				MB_BitStato[192]:=ModBus.MB_MASTER.ReceiveBuffer.Data[3].0; (*Vedi Tabella *)
				MB_BitStato[193]:=ModBus.MB_MASTER.ReceiveBuffer.Data[3].1; (*Vedi Tabella *)
				MB_BitStato[194]:=ModBus.MB_MASTER.ReceiveBuffer.Data[3].2; (*Vedi Tabella *)
				MB_BitStato[195]:=ModBus.MB_MASTER.ReceiveBuffer.Data[3].3; (*Vedi Tabella *)
				MB_BitStato[196]:=ModBus.MB_MASTER.ReceiveBuffer.Data[3].4; (*Vedi Tabella *)
				MB_BitStato[197]:=ModBus.MB_MASTER.ReceiveBuffer.Data[3].5; (*Vedi Tabella *)
				MB_BitStato[198]:=ModBus.MB_MASTER.ReceiveBuffer.Data[3].6; (*Vedi Tabella *)
				MB_BitStato[199]:=ModBus.MB_MASTER.ReceiveBuffer.Data[3].7; (*Vedi Tabella *)
				MB_BitStato[200]:=ModBus.MB_MASTER.ReceiveBuffer.Data[4].0; (*Vedi Tabella *)
				MB_BitStato[201]:=ModBus.MB_MASTER.ReceiveBuffer.Data[4].1; (*Vedi Tabella *)
				MB_BitStato[202]:=ModBus.MB_MASTER.ReceiveBuffer.Data[4].2; (*Vedi Tabella *)
				MB_BitStato[203]:=ModBus.MB_MASTER.ReceiveBuffer.Data[4].3; (*Vedi Tabella *)
				MB_BitStato[204]:=ModBus.MB_MASTER.ReceiveBuffer.Data[4].4; (*Vedi Tabella *)
				MB_BitStato[205]:=ModBus.MB_MASTER.ReceiveBuffer.Data[4].5; (*Vedi Tabella *)
				MB_BitStato[206]:=ModBus.MB_MASTER.ReceiveBuffer.Data[4].6; (*Vedi Tabella *)
				MB_BitStato[207]:=ModBus.MB_MASTER.ReceiveBuffer.Data[4].7; (*Vedi Tabella *)
				MB_BitStato[208]:=ModBus.MB_MASTER.ReceiveBuffer.Data[5].0; (*Vedi Tabella *)
				MB_BitStato[209]:=ModBus.MB_MASTER.ReceiveBuffer.Data[5].1; (*Vedi Tabella *)
				MB_BitStato[210]:=ModBus.MB_MASTER.ReceiveBuffer.Data[5].2; (*Vedi Tabella *)
				MB_BitStato[211]:=ModBus.MB_MASTER.ReceiveBuffer.Data[5].3; (*Vedi Tabella *)
				MB_BitStato[212]:=ModBus.MB_MASTER.ReceiveBuffer.Data[5].4; (*Vedi Tabella *)
				MB_BitStato[213]:=ModBus.MB_MASTER.ReceiveBuffer.Data[5].5; (*Vedi Tabella *)
				MB_BitStato[214]:=ModBus.MB_MASTER.ReceiveBuffer.Data[5].6; (*Vedi Tabella *)
				MB_BitStato[215]:=ModBus.MB_MASTER.ReceiveBuffer.Data[5].7; (*Vedi Tabella *)
				MB_BitStato[216]:=ModBus.MB_MASTER.ReceiveBuffer.Data[6].0; (*Vedi Tabella *)
				MB_BitStato[217]:=ModBus.MB_MASTER.ReceiveBuffer.Data[6].1; (*Vedi Tabella *)
				MB_BitStato[218]:=ModBus.MB_MASTER.ReceiveBuffer.Data[6].2; (*Vedi Tabella *)
				MB_BitStato[219]:=ModBus.MB_MASTER.ReceiveBuffer.Data[6].3; (*Vedi Tabella *)
				MB_BitStato[220]:=ModBus.MB_MASTER.ReceiveBuffer.Data[6].4; (*Vedi Tabella *)
				MB_BitStato[221]:=ModBus.MB_MASTER.ReceiveBuffer.Data[6].5; (*Vedi Tabella *)
				MB_BitStato[222]:=ModBus.MB_MASTER.ReceiveBuffer.Data[6].6; (*Vedi Tabella *)
				MB_BitStato[223]:=ModBus.MB_MASTER.ReceiveBuffer.Data[6].7; (*Vedi Tabella *)
				MB_BitStato[224]:=ModBus.MB_MASTER.ReceiveBuffer.Data[7].0; (*Vedi Tabella *)
				MB_BitStato[225]:=ModBus.MB_MASTER.ReceiveBuffer.Data[7].1; (*Vedi Tabella *)
				MB_BitStato[226]:=ModBus.MB_MASTER.ReceiveBuffer.Data[7].2; (*Vedi Tabella *)
				MB_BitStato[227]:=ModBus.MB_MASTER.ReceiveBuffer.Data[7].3; (*Vedi Tabella *)
				MB_BitStato[228]:=ModBus.MB_MASTER.ReceiveBuffer.Data[7].4; (*Vedi Tabella *)
				MB_BitStato[229]:=ModBus.MB_MASTER.ReceiveBuffer.Data[7].5; (*Vedi Tabella *)
				MB_BitStato[230]:=ModBus.MB_MASTER.ReceiveBuffer.Data[7].6; (*Vedi Tabella *)
				MB_BitStato[231]:=ModBus.MB_MASTER.ReceiveBuffer.Data[7].7; (*Vedi Tabella *)
				MB_BitStato[232]:=ModBus.MB_MASTER.ReceiveBuffer.Data[8].0; (*Vedi Tabella *)
				MB_BitStato[233]:=ModBus.MB_MASTER.ReceiveBuffer.Data[8].1; (*Vedi Tabella *)
				MB_BitStato[234]:=ModBus.MB_MASTER.ReceiveBuffer.Data[8].2; (*Vedi Tabella *)
				MB_BitStato[235]:=ModBus.MB_MASTER.ReceiveBuffer.Data[8].3; (*Vedi Tabella *)
				MB_BitStato[236]:=ModBus.MB_MASTER.ReceiveBuffer.Data[8].4; (*Vedi Tabella *)
				MB_BitStato[237]:=ModBus.MB_MASTER.ReceiveBuffer.Data[8].5; (*Vedi Tabella *)
				MB_BitStato[238]:=ModBus.MB_MASTER.ReceiveBuffer.Data[8].6; (*Vedi Tabella *)
				MB_BitStato[239]:=ModBus.MB_MASTER.ReceiveBuffer.Data[8].7; (*Vedi Tabella *)
				MB_BitStato[240]:=ModBus.MB_MASTER.ReceiveBuffer.Data[9].0; (*Vedi Tabella *)
				MB_BitStato[241]:=ModBus.MB_MASTER.ReceiveBuffer.Data[9].1; (*Vedi Tabella *)
				MB_BitStato[242]:=ModBus.MB_MASTER.ReceiveBuffer.Data[9].2; (*Vedi Tabella *)
				MB_BitStato[243]:=ModBus.MB_MASTER.ReceiveBuffer.Data[9].3; (*Vedi Tabella *)
				MB_BitStato[244]:=ModBus.MB_MASTER.ReceiveBuffer.Data[9].4; (*Vedi Tabella *)
				MB_BitStato[245]:=ModBus.MB_MASTER.ReceiveBuffer.Data[9].5; (*Vedi Tabella *)
				MB_BitStato[246]:=ModBus.MB_MASTER.ReceiveBuffer.Data[9].6; (*Vedi Tabella *)
				MB_BitStato[247]:=ModBus.MB_MASTER.ReceiveBuffer.Data[9].7; (*Vedi Tabella *)
				MB_BitStato[248]:=ModBus.MB_MASTER.ReceiveBuffer.Data[10].0; (*Vedi Tabella *)
				MB_BitStato[249]:=ModBus.MB_MASTER.ReceiveBuffer.Data[10].1; (*Vedi Tabella *)
				MB_BitStato[250]:=ModBus.MB_MASTER.ReceiveBuffer.Data[10].2; (*Vedi Tabella *)
				MB_BitStato[251]:=ModBus.MB_MASTER.ReceiveBuffer.Data[10].3; (*Vedi Tabella *)
				MB_BitStato[252]:=ModBus.MB_MASTER.ReceiveBuffer.Data[10].4; (*Vedi Tabella *)
				MB_BitStato[253]:=ModBus.MB_MASTER.ReceiveBuffer.Data[10].5; (*Vedi Tabella *)
				MB_BitStato[254]:=ModBus.MB_MASTER.ReceiveBuffer.Data[10].6; (*Vedi Tabella *)
				MB_BitStato[255]:=ModBus.MB_MASTER.ReceiveBuffer.Data[10].7; (*Vedi Tabella *)

				state:=140;

			END_IF
		END_IF

	140: (* Rispota Altri paramenti COIL *)
		IF NOT ModBus.MB_Start  THEN

			IF ModBus.MB_MASTER.MB_Error<>0 THEN
				state := 300;
			ELSE
				Modbus.MB_Query.SlaveAddress := Address;
				Modbus.MB_Query.FunctionCode := 2;
				ModBus.MB_Query.Read_StartAddress := 256;	(* richiedo lettura altri Parametri *)
				ModBus.MB_Query.Read_Quantity := 64;
				ModBus.MB_Start := TRUE;

				state:=145;
			END_IF
		END_IF
	145: (* Rispota Altri paramenti *)

		IF NOT ModBus.MB_Start  THEN

			IF ModBus.MB_MASTER.MB_Error<>0 THEN
				state := 300;
			ELSE

				MB_BitStato[256]:=ModBus.MB_MASTER.ReceiveBuffer.Data[3].0; (*Vedi Tabella *)
				MB_BitStato[257]:=ModBus.MB_MASTER.ReceiveBuffer.Data[3].1; (*Vedi Tabella *)
				MB_BitStato[258]:=ModBus.MB_MASTER.ReceiveBuffer.Data[3].2; (*Vedi Tabella *)
				MB_BitStato[259]:=ModBus.MB_MASTER.ReceiveBuffer.Data[3].3; (*Vedi Tabella *)
				MB_BitStato[260]:=ModBus.MB_MASTER.ReceiveBuffer.Data[3].4; (*Vedi Tabella *)
				MB_BitStato[261]:=ModBus.MB_MASTER.ReceiveBuffer.Data[3].5; (*Vedi Tabella *)
				MB_BitStato[262]:=ModBus.MB_MASTER.ReceiveBuffer.Data[3].6; (*Vedi Tabella *)
				MB_BitStato[263]:=ModBus.MB_MASTER.ReceiveBuffer.Data[3].7; (*Vedi Tabella *)
				MB_BitStato[264]:=ModBus.MB_MASTER.ReceiveBuffer.Data[4].0; (*Vedi Tabella *)
				MB_BitStato[265]:=ModBus.MB_MASTER.ReceiveBuffer.Data[4].1; (*Vedi Tabella *)
				MB_BitStato[266]:=ModBus.MB_MASTER.ReceiveBuffer.Data[4].2; (*Vedi Tabella *)
				MB_BitStato[267]:=ModBus.MB_MASTER.ReceiveBuffer.Data[4].3; (*Vedi Tabella *)
				MB_BitStato[268]:=ModBus.MB_MASTER.ReceiveBuffer.Data[4].4; (*Vedi Tabella *)
				MB_BitStato[269]:=ModBus.MB_MASTER.ReceiveBuffer.Data[4].5; (*Vedi Tabella *)
				MB_BitStato[270]:=ModBus.MB_MASTER.ReceiveBuffer.Data[4].6; (*Vedi Tabella *)
				MB_BitStato[271]:=ModBus.MB_MASTER.ReceiveBuffer.Data[4].7; (*Vedi Tabella *)
				MB_BitStato[272]:=ModBus.MB_MASTER.ReceiveBuffer.Data[5].0; (*Vedi Tabella *)
				MB_BitStato[273]:=ModBus.MB_MASTER.ReceiveBuffer.Data[5].1; (*Vedi Tabella *)
				MB_BitStato[274]:=ModBus.MB_MASTER.ReceiveBuffer.Data[5].2; (*Vedi Tabella *)
				MB_BitStato[275]:=ModBus.MB_MASTER.ReceiveBuffer.Data[5].3; (*Vedi Tabella *)
				MB_BitStato[276]:=ModBus.MB_MASTER.ReceiveBuffer.Data[5].4; (*Vedi Tabella *)
				MB_BitStato[277]:=ModBus.MB_MASTER.ReceiveBuffer.Data[5].5; (*Vedi Tabella *)
				MB_BitStato[278]:=ModBus.MB_MASTER.ReceiveBuffer.Data[5].6; (*Vedi Tabella *)
				MB_BitStato[279]:=ModBus.MB_MASTER.ReceiveBuffer.Data[5].7; (*Vedi Tabella *)
				MB_BitStato[280]:=ModBus.MB_MASTER.ReceiveBuffer.Data[6].0; (*Vedi Tabella *)
				MB_BitStato[281]:=ModBus.MB_MASTER.ReceiveBuffer.Data[6].1; (*Vedi Tabella *)
				MB_BitStato[282]:=ModBus.MB_MASTER.ReceiveBuffer.Data[6].2; (*Vedi Tabella *)
				MB_BitStato[283]:=ModBus.MB_MASTER.ReceiveBuffer.Data[6].3; (*Vedi Tabella *)
				MB_BitStato[284]:=ModBus.MB_MASTER.ReceiveBuffer.Data[6].4; (*Vedi Tabella *)
				MB_BitStato[285]:=ModBus.MB_MASTER.ReceiveBuffer.Data[6].5; (*Vedi Tabella *)
				MB_BitStato[286]:=ModBus.MB_MASTER.ReceiveBuffer.Data[6].6; (*Vedi Tabella *)
				MB_BitStato[287]:=ModBus.MB_MASTER.ReceiveBuffer.Data[6].7; (*Vedi Tabella *)
				MB_BitStato[288]:=ModBus.MB_MASTER.ReceiveBuffer.Data[7].0; (*Vedi Tabella *)
				MB_BitStato[289]:=ModBus.MB_MASTER.ReceiveBuffer.Data[7].1; (*Vedi Tabella *)
				MB_BitStato[290]:=ModBus.MB_MASTER.ReceiveBuffer.Data[7].2; (*Vedi Tabella *)
				MB_BitStato[291]:=ModBus.MB_MASTER.ReceiveBuffer.Data[7].3; (*Vedi Tabella *)
				MB_BitStato[292]:=ModBus.MB_MASTER.ReceiveBuffer.Data[7].4; (*Vedi Tabella *)
				MB_BitStato[293]:=ModBus.MB_MASTER.ReceiveBuffer.Data[7].5; (*Vedi Tabella *)
				MB_BitStato[294]:=ModBus.MB_MASTER.ReceiveBuffer.Data[7].6; (*Vedi Tabella *)
				MB_BitStato[295]:=ModBus.MB_MASTER.ReceiveBuffer.Data[7].7; (*Vedi Tabella *)
				MB_BitStato[296]:=ModBus.MB_MASTER.ReceiveBuffer.Data[8].0; (*Vedi Tabella *)
				MB_BitStato[297]:=ModBus.MB_MASTER.ReceiveBuffer.Data[8].1; (*Vedi Tabella *)
				MB_BitStato[298]:=ModBus.MB_MASTER.ReceiveBuffer.Data[8].2; (*Vedi Tabella *)
				MB_BitStato[299]:=ModBus.MB_MASTER.ReceiveBuffer.Data[8].3; (*Vedi Tabella *)
				MB_BitStato[300]:=ModBus.MB_MASTER.ReceiveBuffer.Data[8].4; (*Vedi Tabella *)
				MB_BitStato[301]:=ModBus.MB_MASTER.ReceiveBuffer.Data[8].5; (*Vedi Tabella *)
				MB_BitStato[302]:=ModBus.MB_MASTER.ReceiveBuffer.Data[8].6; (*Vedi Tabella *)
				MB_BitStato[303]:=ModBus.MB_MASTER.ReceiveBuffer.Data[8].7; (*Vedi Tabella *)
				MB_BitStato[304]:=ModBus.MB_MASTER.ReceiveBuffer.Data[9].0; (*Vedi Tabella *)
				MB_BitStato[305]:=ModBus.MB_MASTER.ReceiveBuffer.Data[9].1; (*Vedi Tabella *)
				MB_BitStato[306]:=ModBus.MB_MASTER.ReceiveBuffer.Data[9].2; (*Vedi Tabella *)
				MB_BitStato[307]:=ModBus.MB_MASTER.ReceiveBuffer.Data[9].3; (*Vedi Tabella *)
				MB_BitStato[308]:=ModBus.MB_MASTER.ReceiveBuffer.Data[9].4; (*Vedi Tabella *)
				MB_BitStato[309]:=ModBus.MB_MASTER.ReceiveBuffer.Data[9].5; (*Vedi Tabella *)
				MB_BitStato[310]:=ModBus.MB_MASTER.ReceiveBuffer.Data[9].6; (*Vedi Tabella *)
				MB_BitStato[311]:=ModBus.MB_MASTER.ReceiveBuffer.Data[9].7; (*Vedi Tabella *)
				MB_BitStato[312]:=ModBus.MB_MASTER.ReceiveBuffer.Data[10].0; (*Vedi Tabella *)
				MB_BitStato[313]:=ModBus.MB_MASTER.ReceiveBuffer.Data[10].1; (*Vedi Tabella *)
				MB_BitStato[314]:=ModBus.MB_MASTER.ReceiveBuffer.Data[10].2; (*Vedi Tabella *)
				MB_BitStato[315]:=ModBus.MB_MASTER.ReceiveBuffer.Data[10].3; (*Vedi Tabella *)
				MB_BitStato[316]:=ModBus.MB_MASTER.ReceiveBuffer.Data[10].4; (*Vedi Tabella *)
				MB_BitStato[317]:=ModBus.MB_MASTER.ReceiveBuffer.Data[10].5; (*Vedi Tabella *)
				MB_BitStato[318]:=ModBus.MB_MASTER.ReceiveBuffer.Data[10].6; (*Vedi Tabella *)
				MB_BitStato[319]:=ModBus.MB_MASTER.ReceiveBuffer.Data[10].7; (*Vedi Tabella *)

				state:=160;

			END_IF
		END_IF

	160: (* Rispota Altri paramenti COIL *)
		IF NOT ModBus.MB_Start  THEN

			IF ModBus.MB_MASTER.MB_Error<>0 THEN
				state := 300;
			ELSE
				Modbus.MB_Query.SlaveAddress := Address;
				Modbus.MB_Query.FunctionCode := 2;
				ModBus.MB_Query.Read_StartAddress := 320;	(* richiedo lettura altri Parametri *)
				ModBus.MB_Query.Read_Quantity := 64;
				ModBus.MB_Start := TRUE;

				state:=165;
			END_IF
		END_IF
	165: (* Rispota Altri paramenti *)

		IF NOT ModBus.MB_Start  THEN

			IF ModBus.MB_MASTER.MB_Error<>0 THEN
				state := 300;
			ELSE

				MB_BitStato[320]:=ModBus.MB_MASTER.ReceiveBuffer.Data[3].0; (*Vedi Tabella *)
				MB_BitStato[321]:=ModBus.MB_MASTER.ReceiveBuffer.Data[3].1; (*Vedi Tabella *)
				MB_BitStato[322]:=ModBus.MB_MASTER.ReceiveBuffer.Data[3].2; (*Vedi Tabella *)
				MB_BitStato[323]:=ModBus.MB_MASTER.ReceiveBuffer.Data[3].3; (*Vedi Tabella *)
				MB_BitStato[324]:=ModBus.MB_MASTER.ReceiveBuffer.Data[3].4; (*Vedi Tabella *)
				MB_BitStato[325]:=ModBus.MB_MASTER.ReceiveBuffer.Data[3].5; (*Vedi Tabella *)
				MB_BitStato[326]:=ModBus.MB_MASTER.ReceiveBuffer.Data[3].6; (*Vedi Tabella *)
				MB_BitStato[327]:=ModBus.MB_MASTER.ReceiveBuffer.Data[3].7; (*Vedi Tabella *)
				MB_BitStato[328]:=ModBus.MB_MASTER.ReceiveBuffer.Data[4].0; (*Vedi Tabella *)
				MB_BitStato[329]:=ModBus.MB_MASTER.ReceiveBuffer.Data[4].1; (*Vedi Tabella *)
				MB_BitStato[330]:=ModBus.MB_MASTER.ReceiveBuffer.Data[4].2; (*Vedi Tabella *)
				MB_BitStato[331]:=ModBus.MB_MASTER.ReceiveBuffer.Data[4].3; (*Vedi Tabella *)
				MB_BitStato[332]:=ModBus.MB_MASTER.ReceiveBuffer.Data[4].4; (*Vedi Tabella *)
				MB_BitStato[333]:=ModBus.MB_MASTER.ReceiveBuffer.Data[4].5; (*Vedi Tabella *)
				MB_BitStato[334]:=ModBus.MB_MASTER.ReceiveBuffer.Data[4].6; (*Vedi Tabella *)
				MB_BitStato[335]:=ModBus.MB_MASTER.ReceiveBuffer.Data[4].7; (*Vedi Tabella *)
				MB_BitStato[336]:=ModBus.MB_MASTER.ReceiveBuffer.Data[5].0; (*Vedi Tabella *)
				MB_BitStato[337]:=ModBus.MB_MASTER.ReceiveBuffer.Data[5].1; (*Vedi Tabella *)
				MB_BitStato[338]:=ModBus.MB_MASTER.ReceiveBuffer.Data[5].2; (*Vedi Tabella *)
				MB_BitStato[339]:=ModBus.MB_MASTER.ReceiveBuffer.Data[5].3; (*Vedi Tabella *)
				MB_BitStato[340]:=ModBus.MB_MASTER.ReceiveBuffer.Data[5].4; (*Vedi Tabella *)
				MB_BitStato[341]:=ModBus.MB_MASTER.ReceiveBuffer.Data[5].5; (*Vedi Tabella *)
				MB_BitStato[342]:=ModBus.MB_MASTER.ReceiveBuffer.Data[5].6; (*Vedi Tabella *)
				MB_BitStato[343]:=ModBus.MB_MASTER.ReceiveBuffer.Data[5].7; (*Vedi Tabella *)
				MB_BitStato[344]:=ModBus.MB_MASTER.ReceiveBuffer.Data[6].0; (*Vedi Tabella *)
				MB_BitStato[345]:=ModBus.MB_MASTER.ReceiveBuffer.Data[6].1; (*Vedi Tabella *)
				MB_BitStato[346]:=ModBus.MB_MASTER.ReceiveBuffer.Data[6].2; (*Vedi Tabella *)
				MB_BitStato[347]:=ModBus.MB_MASTER.ReceiveBuffer.Data[6].3; (*Vedi Tabella *)
				MB_BitStato[348]:=ModBus.MB_MASTER.ReceiveBuffer.Data[6].4; (*Vedi Tabella *)
				MB_BitStato[349]:=ModBus.MB_MASTER.ReceiveBuffer.Data[6].5; (*Vedi Tabella *)
				MB_BitStato[350]:=ModBus.MB_MASTER.ReceiveBuffer.Data[6].6; (*Vedi Tabella *)
				MB_BitStato[351]:=ModBus.MB_MASTER.ReceiveBuffer.Data[6].7; (*Vedi Tabella *)
				MB_BitStato[352]:=ModBus.MB_MASTER.ReceiveBuffer.Data[7].0; (*Vedi Tabella *)
				MB_BitStato[353]:=ModBus.MB_MASTER.ReceiveBuffer.Data[7].1; (*Vedi Tabella *)
				MB_BitStato[354]:=ModBus.MB_MASTER.ReceiveBuffer.Data[7].2; (*Vedi Tabella *)
				MB_BitStato[355]:=ModBus.MB_MASTER.ReceiveBuffer.Data[7].3; (*Vedi Tabella *)
				MB_BitStato[356]:=ModBus.MB_MASTER.ReceiveBuffer.Data[7].4; (*Vedi Tabella *)
				MB_BitStato[357]:=ModBus.MB_MASTER.ReceiveBuffer.Data[7].5; (*Vedi Tabella *)
	(*			MB_BitStato[359]:=ModBus.MB_MASTER.ReceiveBuffer.Data[7].6; (*Vedi Tabella *)
				MB_BitStato[360]:=ModBus.MB_MASTER.ReceiveBuffer.Data[7].7; (*Vedi Tabella *)
				MB_BitStato[40]:=ModBus.MB_MASTER.ReceiveBuffer.Data[8].0; (*Vedi Tabella *)
				MB_BitStato[41]:=ModBus.MB_MASTER.ReceiveBuffer.Data[8].1; (*Vedi Tabella *)
				MB_BitStato[42]:=ModBus.MB_MASTER.ReceiveBuffer.Data[8].2; (*Vedi Tabella *)
				MB_BitStato[43]:=ModBus.MB_MASTER.ReceiveBuffer.Data[8].3; (*Vedi Tabella *)
				MB_BitStato[44]:=ModBus.MB_MASTER.ReceiveBuffer.Data[8].4; (*Vedi Tabella *)
				MB_BitStato[45]:=ModBus.MB_MASTER.ReceiveBuffer.Data[8].5; (*Vedi Tabella *)
				MB_BitStato[46]:=ModBus.MB_MASTER.ReceiveBuffer.Data[8].6; (*Vedi Tabella *)
				MB_BitStato[47]:=ModBus.MB_MASTER.ReceiveBuffer.Data[8].7; (*Vedi Tabella *)
				MB_BitStato[48]:=ModBus.MB_MASTER.ReceiveBuffer.Data[9].0; (*Vedi Tabella *)
				MB_BitStato[49]:=ModBus.MB_MASTER.ReceiveBuffer.Data[9].1; (*Vedi Tabella *)
				MB_BitStato[50]:=ModBus.MB_MASTER.ReceiveBuffer.Data[9].2; (*Vedi Tabella *)
				MB_BitStato[51]:=ModBus.MB_MASTER.ReceiveBuffer.Data[9].3; (*Vedi Tabella *)
				MB_BitStato[52]:=ModBus.MB_MASTER.ReceiveBuffer.Data[9].4; (*Vedi Tabella *)
				MB_BitStato[53]:=ModBus.MB_MASTER.ReceiveBuffer.Data[9].5; (*Vedi Tabella *)
				MB_BitStato[54]:=ModBus.MB_MASTER.ReceiveBuffer.Data[9].6; (*Vedi Tabella *)
				MB_BitStato[55]:=ModBus.MB_MASTER.ReceiveBuffer.Data[9].7; (*Vedi Tabella *)
				MB_BitStato[56]:=ModBus.MB_MASTER.ReceiveBuffer.Data[10].0; (*Vedi Tabella *)
				MB_BitStato[57]:=ModBus.MB_MASTER.ReceiveBuffer.Data[10].1; (*Vedi Tabella *)
				MB_BitStato[58]:=ModBus.MB_MASTER.ReceiveBuffer.Data[10].2; (*Vedi Tabella *)
				MB_BitStato[59]:=ModBus.MB_MASTER.ReceiveBuffer.Data[10].3; (*Vedi Tabella *)
				MB_BitStato[60]:=ModBus.MB_MASTER.ReceiveBuffer.Data[10].4; (*Vedi Tabella *)
				MB_BitStato[61]:=ModBus.MB_MASTER.ReceiveBuffer.Data[10].5; (*Vedi Tabella *)
				MB_BitStato[62]:=ModBus.MB_MASTER.ReceiveBuffer.Data[10].6; (*Vedi Tabella *)
				MB_BitStato[63]:=ModBus.MB_MASTER.ReceiveBuffer.Data[10].7; (*Vedi Tabella *)
*)
				state:=170;

			END_IF
		END_IF





	170: (* Rispota Altri paramenti COIL *)
		IF NOT ModBus.MB_Start  THEN

			IF ModBus.MB_MASTER.MB_Error<>0 THEN
				state := 300;
			ELSE
				Modbus.MB_Query.SlaveAddress := Address;
				Modbus.MB_Query.FunctionCode := 1;
				ModBus.MB_Query.Read_StartAddress := 0;	(* richiedo lettura altri Parametri *)
				ModBus.MB_Query.Read_Quantity := 64;
				ModBus.MB_Start := TRUE;

				state:=171;
			END_IF
		END_IF
	171: (* Rispota Altri paramenti *)

		IF NOT ModBus.MB_Start  THEN

			IF ModBus.MB_MASTER.MB_Error<>0 THEN
				state := 300;
			ELSE

				MB_BitStatoCoil[0]:=ModBus.MB_MASTER.ReceiveBuffer.Data[3].0; (*Vedi Tabella *)
				MB_BitStatoCoil[1]:=ModBus.MB_MASTER.ReceiveBuffer.Data[3].1; (*Vedi Tabella *)
				MB_BitStatoCoil[2]:=ModBus.MB_MASTER.ReceiveBuffer.Data[3].2; (*Vedi Tabella *)
				MB_BitStatoCoil[3]:=ModBus.MB_MASTER.ReceiveBuffer.Data[3].3; (*Vedi Tabella *)
				MB_BitStatoCoil[4]:=ModBus.MB_MASTER.ReceiveBuffer.Data[3].4; (*Vedi Tabella *)
				MB_BitStatoCoil[5]:=ModBus.MB_MASTER.ReceiveBuffer.Data[3].5; (*Vedi Tabella *)
				MB_BitStatoCoil[6]:=ModBus.MB_MASTER.ReceiveBuffer.Data[3].6; (*Vedi Tabella *)
				MB_BitStatoCoil[7]:=ModBus.MB_MASTER.ReceiveBuffer.Data[3].7; (*Vedi Tabella *)
				MB_BitStatoCoil[8]:=ModBus.MB_MASTER.ReceiveBuffer.Data[4].0; (*Vedi Tabella *)
				MB_BitStatoCoil[9]:=ModBus.MB_MASTER.ReceiveBuffer.Data[4].1; (*Vedi Tabella *)
				MB_BitStatoCoil[10]:=ModBus.MB_MASTER.ReceiveBuffer.Data[4].2; (*Vedi Tabella *)
				MB_BitStatoCoil[11]:=ModBus.MB_MASTER.ReceiveBuffer.Data[4].3; (*Vedi Tabella *)
				MB_BitStatoCoil[12]:=ModBus.MB_MASTER.ReceiveBuffer.Data[4].4; (*Vedi Tabella *)
				MB_BitStatoCoil[13]:=ModBus.MB_MASTER.ReceiveBuffer.Data[4].5; (*Vedi Tabella *)
				MB_BitStatoCoil[14]:=ModBus.MB_MASTER.ReceiveBuffer.Data[4].6; (*Vedi Tabella *)
				MB_BitStatoCoil[15]:=ModBus.MB_MASTER.ReceiveBuffer.Data[4].7; (*Vedi Tabella *)
				MB_BitStatoCoil[16]:=ModBus.MB_MASTER.ReceiveBuffer.Data[5].0; (*Vedi Tabella *)
				MB_BitStatoCoil[17]:=ModBus.MB_MASTER.ReceiveBuffer.Data[5].1; (*Vedi Tabella *)
				MB_BitStatoCoil[18]:=ModBus.MB_MASTER.ReceiveBuffer.Data[5].2; (*Vedi Tabella *)
				MB_BitStatoCoil[19]:=ModBus.MB_MASTER.ReceiveBuffer.Data[5].3; (*Vedi Tabella *)
				MB_BitStatoCoil[20]:=ModBus.MB_MASTER.ReceiveBuffer.Data[5].4; (*Vedi Tabella *)
				MB_BitStatoCoil[21]:=ModBus.MB_MASTER.ReceiveBuffer.Data[5].5; (*Vedi Tabella *)
				MB_BitStatoCoil[22]:=ModBus.MB_MASTER.ReceiveBuffer.Data[5].6; (*Vedi Tabella *)
				MB_BitStatoCoil[23]:=ModBus.MB_MASTER.ReceiveBuffer.Data[5].7; (*Vedi Tabella *)
				MB_BitStatoCoil[24]:=ModBus.MB_MASTER.ReceiveBuffer.Data[6].0; (*Vedi Tabella *)
				MB_BitStatoCoil[25]:=ModBus.MB_MASTER.ReceiveBuffer.Data[6].1; (*Vedi Tabella *)
				MB_BitStatoCoil[26]:=ModBus.MB_MASTER.ReceiveBuffer.Data[6].2; (*Vedi Tabella *)
				MB_BitStatoCoil[27]:=ModBus.MB_MASTER.ReceiveBuffer.Data[6].3; (*Vedi Tabella *)
				MB_BitStatoCoil[28]:=ModBus.MB_MASTER.ReceiveBuffer.Data[6].4; (*Vedi Tabella *)
				MB_BitStatoCoil[29]:=ModBus.MB_MASTER.ReceiveBuffer.Data[6].5; (*Vedi Tabella *)
				MB_BitStatoCoil[30]:=ModBus.MB_MASTER.ReceiveBuffer.Data[6].6; (*Vedi Tabella *)
				MB_BitStatoCoil[31]:=ModBus.MB_MASTER.ReceiveBuffer.Data[6].7; (*Vedi Tabella *)
				MB_BitStatoCoil[32]:=ModBus.MB_MASTER.ReceiveBuffer.Data[7].0; (*Vedi Tabella *)
				MB_BitStatoCoil[33]:=ModBus.MB_MASTER.ReceiveBuffer.Data[7].1; (*Vedi Tabella *)
				MB_BitStatoCoil[34]:=ModBus.MB_MASTER.ReceiveBuffer.Data[7].2; (*Vedi Tabella *)
				MB_BitStatoCoil[35]:=ModBus.MB_MASTER.ReceiveBuffer.Data[7].3; (*Vedi Tabella *)
				MB_BitStatoCoil[36]:=ModBus.MB_MASTER.ReceiveBuffer.Data[7].4; (*Vedi Tabella *)
				MB_BitStatoCoil[37]:=ModBus.MB_MASTER.ReceiveBuffer.Data[7].5; (*Vedi Tabella *)
				MB_BitStatoCoil[38]:=ModBus.MB_MASTER.ReceiveBuffer.Data[7].6; (*Vedi Tabella *)
				MB_BitStatoCoil[39]:=ModBus.MB_MASTER.ReceiveBuffer.Data[7].7; (*Vedi Tabella *)
				MB_BitStatoCoil[40]:=ModBus.MB_MASTER.ReceiveBuffer.Data[8].0; (*Vedi Tabella *)
				MB_BitStatoCoil[41]:=ModBus.MB_MASTER.ReceiveBuffer.Data[8].1; (*Vedi Tabella *)
				MB_BitStatoCoil[42]:=ModBus.MB_MASTER.ReceiveBuffer.Data[8].2; (*Vedi Tabella *)
				MB_BitStatoCoil[43]:=ModBus.MB_MASTER.ReceiveBuffer.Data[8].3; (*Vedi Tabella *)
				MB_BitStatoCoil[44]:=ModBus.MB_MASTER.ReceiveBuffer.Data[8].4; (*Vedi Tabella *)
				MB_BitStatoCoil[45]:=ModBus.MB_MASTER.ReceiveBuffer.Data[8].5; (*Vedi Tabella *)
				MB_BitStatoCoil[46]:=ModBus.MB_MASTER.ReceiveBuffer.Data[8].6; (*Vedi Tabella *)
				MB_BitStatoCoil[47]:=ModBus.MB_MASTER.ReceiveBuffer.Data[8].7; (*Vedi Tabella *)
				MB_BitStatoCoil[48]:=ModBus.MB_MASTER.ReceiveBuffer.Data[9].0; (*Vedi Tabella *)
				MB_BitStatoCoil[49]:=ModBus.MB_MASTER.ReceiveBuffer.Data[9].1; (*Vedi Tabella *)
				MB_BitStatoCoil[50]:=ModBus.MB_MASTER.ReceiveBuffer.Data[9].2; (*Vedi Tabella *)
				MB_BitStatoCoil[51]:=ModBus.MB_MASTER.ReceiveBuffer.Data[9].3; (*Vedi Tabella *)
				MB_BitStatoCoil[52]:=ModBus.MB_MASTER.ReceiveBuffer.Data[9].4; (*Vedi Tabella *)
				MB_BitStatoCoil[53]:=ModBus.MB_MASTER.ReceiveBuffer.Data[9].5; (*Vedi Tabella *)
				MB_BitStatoCoil[54]:=ModBus.MB_MASTER.ReceiveBuffer.Data[9].6; (*Vedi Tabella *)
				MB_BitStatoCoil[55]:=ModBus.MB_MASTER.ReceiveBuffer.Data[9].7; (*Vedi Tabella *)
				MB_BitStatoCoil[56]:=ModBus.MB_MASTER.ReceiveBuffer.Data[10].0; (*Vedi Tabella *)
				MB_BitStatoCoil[57]:=ModBus.MB_MASTER.ReceiveBuffer.Data[10].1; (*Vedi Tabella *)
				MB_BitStatoCoil[58]:=ModBus.MB_MASTER.ReceiveBuffer.Data[10].2; (*Vedi Tabella *)
				MB_BitStatoCoil[59]:=ModBus.MB_MASTER.ReceiveBuffer.Data[10].3; (*Vedi Tabella *)
				MB_BitStatoCoil[60]:=ModBus.MB_MASTER.ReceiveBuffer.Data[10].4; (*Vedi Tabella *)
				MB_BitStatoCoil[61]:=ModBus.MB_MASTER.ReceiveBuffer.Data[10].5; (*Vedi Tabella *)
				MB_BitStatoCoil[62]:=ModBus.MB_MASTER.ReceiveBuffer.Data[10].6; (*Vedi Tabella *)
				MB_BitStatoCoil[63]:=ModBus.MB_MASTER.ReceiveBuffer.Data[10].7; (*Vedi Tabella *)
				MB_BitStatoCoil[64]:=ModBus.MB_MASTER.ReceiveBuffer.Data[11].0; (*Vedi Tabella *)
				MB_BitStatoCoil[65]:=ModBus.MB_MASTER.ReceiveBuffer.Data[11].1; (*Vedi Tabella *)
				MB_BitStatoCoil[66]:=ModBus.MB_MASTER.ReceiveBuffer.Data[1].2; (*Vedi Tabella *)
				MB_BitStatoCoil[67]:=ModBus.MB_MASTER.ReceiveBuffer.Data[11].3; (*Vedi Tabella *)
				MB_BitStatoCoil[68]:=ModBus.MB_MASTER.ReceiveBuffer.Data[11].4; (*Vedi Tabella *)
				MB_BitStatoCoil[69]:=ModBus.MB_MASTER.ReceiveBuffer.Data[11].5; (*Vedi Tabella *)
				MB_BitStatoCoil[70]:=ModBus.MB_MASTER.ReceiveBuffer.Data[11].6; (*Vedi Tabella *)
				MB_BitStatoCoil[71]:=ModBus.MB_MASTER.ReceiveBuffer.Data[11].7; (*Vedi Tabella *)
				state:=200;

			END_IF
		END_IF














		200:    (* Scrittura BOOL - COIL o WORD *)
		IF NOT ModBus.MB_Start THEN
			IF ModBus.MB_MASTER.MB_Error<>0 THEN (*OR ModBus.MB_MASTER.MB_Error<>0 THEN*)
				state := 300;
			ELSE
				IF ScriviMB THEN
					IF Test_ScriviCoil THEN
						Modbus.MB_Query.FunctionCode := 5;
					ELSE
						Modbus.MB_Query.FunctionCode := 6;
					END_IF
					Modbus.MB_Query.SlaveAddress := Address;
					ModBus.MB_Query.Write_StartAddress := test_Address;
					ModBus.MB_Query.Write_Quantity :=1;
					ModBus.MB_Query.Write_Data[0] := test_Write;
					ModBus.MB_Start := TRUE;
						IF Test_ScriviCoil THEN
							IF 	MB_BitStatoCoil[test_Address]=WORD_TO_BOOL(test_Write) THEN
								ScriviMB:=FALSE;
							END_IF
						ELSE
							IF 	MB_RegistriHoldingLetti[test_Address]=test_Write THEN
								ScriviMB:=FALSE;
							END_IF
						END_IF
					state := 295;
				ELSE
					state := 295;
				END_IF
			END_IF
		END_IF



		295:
		IF NOT ModBus.MB_Start THEN
			IF ModBus.MB_MASTER.MB_Error<>0 THEN (*OR ModBus.MB_MASTER.MB_Error<>0 THEN*)
				state := 300;
			ELSE
				IF fModbusAlr THEN fModbusAlr := FALSE; END_IF
				NodoDaInterrogareANZ:=Address+1;
				InibiscoModbusANZ:=FALSE;
				retryErr := 0;
				retry := 0;
				state := 0;
					IF fModbusAlr=FALSE AND ErroreComuModBus=TRUE THEN
						LogEv(EL_Log,EO_CHI,ID,62,'ComunicazioneModBus_OK');
						ErroreComuModBus := FALSE;
				(*	WarningCtr := SEL(WarningCtr=0, WarningCtr-1, 0); *)
					END_IF


			END_IF
		END_IF



	(**** CHECK MODBUS ERROR ****)
	300: 	(* Release MODBUS *)
			InibiscoModbusMB1:=FALSE;
			(* Retries *)
			retry:=retry+1;
			IF retry>3 THEN
				retry:=0;

				(* Verify if slave is dead *)
				IF retryErr < retryErrMaX THEN
					retryErr := retryErr + 1;
				ELSE
					fModbusAlr := TRUE;
					(* Verify ModBus error	*)

					IF fModbusAlr AND ErroreComuModBus=FALSE THEN
						LogEv(EL_Alarm,EO_CHI,ID,61,CONCAT('ErroreModbus_',INT_TO_STRING(ModBus.MB_MASTER.MB_Error)));
						ErroreComuModBus := TRUE;
					END_IF
				END_IF

				END_IF
			Refresh_Now := FALSE;
			InibiscoModbusMB1:=FALSE;
			NodoDaInterrogareMB1:=Address;
			state:=0;
END_CASE




(* Controllo Time Out Ciclo ModBus *)

TimeOutModBus(In:=state<>0,PT:=t#30s);
IF TimeOutModBus.Q THEN
	State:=0;
	Refresh_Now:=TRUE;  (* Rilancio la lettura del nodo *)
	IF MODBUS.MB_Lock=TRUE THEN MODBUS.MB_Lock:=FALSE;END_IF
	IF InibiscoModbusMB1=TRUE THEN InibiscoModbusMB1:=FALSE;END_IF
END_IF
END_ACTION

(* POU Plant_Objects/obj_UTA_02, ST *)
FUNCTION_BLOCK obj_UTA_02
VAR_INPUT
	ID				: BYTE;

	UTA_ST : BOOL;
	UTA_CentrAL : BOOL;
	UTA_AUTO:BOOL:=TRUE;

	(* Physical inputs (Force) *)
	UTA_RUN_REQ		: BOOL; (* External run request (no heat or cold requested) *)
	UTA_STOP_REQ	: BOOL; (* External stop request (has priority over RUN signals!) *)



END_VAR
VAR_OUTPUT

END_VAR
VAR

	Status_Log		: WORD;
	Status_Vis		: DWORD;


	AllarmeScattoTermico: BOOL;
	AlarmHw		:	FLT_TAP := (INITEV:=FALSE);

END_VAR
(* Hardware alarm (physical input *)
AlarmHw(IN:=UTA_CentrAL);

IF AlarmHw.EVH THEN
	LogEv(EL_Alarm,EO_UTA,ID,3,'UTA_Riarmato');
	AllarmeScattoTermico := FALSE;
END_IF

IF AlarmHw.EVL THEN
	LogEv(EL_Log,EO_UTA,ID,4,'AllarmeUTA');
	AllarmeScattoTermico := TRUE;
END_IF








(* segnalazione Allarme *)
IF AllarmeScattoTermico  THEN
	Status_Log := 2;
	Status_Vis := COLOR_RED;

ELSE
	Status_Log := 0;
	Status_Vis := COLOR_GREEN;
END_IF
END_FUNCTION_BLOCK
ACTION AddLogData:
Logger.s1:=INSERT('&UTA=',BYTE_TO_STRING(ID),4);
IF ID<10 THEN Logger.s1:=INSERT(Logger.s1,'0',4); END_IF

Logger.s1:=CONCAT(Logger.s1,SEL(UTA_ST,'0','100'));		Logger.s1:=CONCAT(Logger.s1,';');

Logger.s1:=CONCAT(Logger.s1,WORD_TO_STRING(Status_Log));
Logger.s1:=CONCAT(Logger.s1,';');
Logger.s1:=CONCAT(Logger.s1,SEL(UTA_RUN_REQ,'0','100'));
Logger.s1:=CONCAT(Logger.s1,';');
Logger.s1:=CONCAT(Logger.s1,SEL(UTA_STOP_REQ,'0','100'));

Logger.s1:=CONCAT(Logger.s1,';');
Logger.s1:=CONCAT(Logger.s1,SEL(UTA_AUTO,'1','0'));


ADDSTRING(ADR(Logger.TData), ADR(Logger.s1), Logger.TLen);
END_ACTION

(* POU Plant_Objects/obj_ZTHL_01, ST *)
FUNCTION_BLOCK obj_ZTHL_01
(* === ZIGBEE AMBIENT SENSORS MT-200 ===
   v1.0[07/05/05] - Create
*)
VAR CONSTANT
	LQI_Threshold		:	WORD := 100;		(* Zigbee link quality minimum value *)
	LowBattVoltage		:	WORD := 270;		(* Battery is considered low when reaches 1.35V each *)
END_VAR
VAR_INPUT
	(* Settings *)
	ID				: BYTE;
	Address			: BYTE;

(*	Refresh_Period	: TIME:=t#5m;
	(* Controls *)
	Refresh_Auto	: BOOL:=TRUE; (* Enable automatic refresh *)*)

	(* Modbus *)
	Refresh_Now	:	BOOL;	(* Start immediately modbus state machine *)
	retryErrMax	:	BYTE := 2;

	(* Limits *)
	Tmin			: INT := 50;
	Tmax			: INT := 400;
END_VAR
VAR_IN_OUT
	(* Interface *)
	ModBus		:obj_MODBUS;

END_VAR
VAR_OUTPUT
	(* Status *)
	Status_Log		: BYTE;
	Status_Vis 		: DWORD;
END_VAR
VAR


	state		:	INT;
	retry		:	BYTE;
	retryErr	:	BYTE;
	ReadTmr		:	TON := (PT:=T#5s);
	fModbusAlr:BOOL;


	AlarmCtr		: BYTE;
	WarningCtr		: BYTE;

	id_locale: BYTE;

	MB_RegistriLetti: ARRAY [0..20] OF INT;

	Quality			: FLT_EVENT;
	Battery			: FLT_EVENT;
	Temperature		: FLT_EVENT := (INITEV:=FALSE);
	Alarm			: FLT_EVENT;

	ERR				: BOOL;
	fLQI			: BOOL;
	fBatt			: BOOL;
	fTemp			: BOOL;

	StatusOK		: BYTE;			(* 0: Status OK, >=1: Alarm and/or warning		Incremented by 1 when Alarm or Wrn occurs,
																					decremented by 1 when restored	*)
	TimeOutModBus: TON;
	ErroreComuModBus: BOOL;

	VerificaFuctionCode: INT;
	VerificaNodoLetto: INT;


END_VAR
(* stato creato per potere interrogare il nodo corretto *)
id_locale:=ID;

Stm();

checkAlarm();
END_FUNCTION_BLOCK
ACTION AddLogData:
Logger.s1:=INSERT('&ZTHL=',BYTE_TO_STRING(ID),5);
IF ID<10 THEN Logger.s1:=INSERT(Logger.s1,'0',5); END_IF

Logger.s1:=CONCAT(Logger.s1,INT_TO_STRING(MB_RegistriLetti[3]));	(* Livello segnale radio dell'ultimo messaggio ricevuto dal dispositivo  *)
Logger.s1:=CONCAT(Logger.s1,';');
Logger.s1:=CONCAT(Logger.s1,INT_TO_STRING(MB_RegistriLetti[6]));	(* Temperatura (in decimi di grado centigrado)  *)
Logger.s1:=CONCAT(Logger.s1,';');
Logger.s1:=CONCAT(Logger.s1,INT_TO_STRING(MB_RegistriLetti[8]));	(* Umidità (espressa in % Umidità Relativa)  *)
Logger.s1:=CONCAT(Logger.s1,';');
Logger.s1:=CONCAT(Logger.s1,INT_TO_STRING(MB_RegistriLetti[5]));	(* Valore efficace Luce (espressa in Lux)  *)
Logger.s1:=CONCAT(Logger.s1,';');
Logger.s1:=CONCAT(Logger.s1,INT_TO_STRING(MB_RegistriLetti[4]));	(* Livello di Batteria (in millesimi di volt) *)
Logger.s1:=CONCAT(Logger.s1,';');

Logger.s1:=CONCAT(Logger.s1,BYTE_TO_STRING(Status_Log));
ADDSTRING(ADR(Logger.TData), ADR(Logger.s1), Logger.TLen);
END_ACTION
ACTION CheckAlarm:
(**** GEstione Log ad Evento *****)


(* (MB_RegistriLetti[3]) check Livello segnale radio dell'ultimo messaggio ricevuto dal dispositivo *)

IF (MB_RegistriLetti[3]) < LQI_Threshold THEN
	fLQI := FALSE;
	ERR := TRUE;
ELSE
	fLQI := TRUE;
	ERR := FALSE;
END_IF

Quality(IN:=fLQI);

IF Quality.EVL THEN
	LogEv(SEL((MB_RegistriLetti[3])<>0,EL_Alarm,EL_Wrn),EO_ZTHL,ID,SEL((MB_RegistriLetti[3])<>0,7,2),WORD_TO_STRING((MB_RegistriLetti[3])));
	Status_Log := SEL((MB_RegistriLetti[3])<>0,2,1);
	StatusOK := StatusOK + 1;
END_IF

IF Quality.EVH THEN StatusOK := SEL(StatusOK=0, StatusOK-1, 0); END_IF

(* If probe (node) is present proceed checking other warnings, otherwise don't transmit anything *)
IF (MB_RegistriLetti[3]) <> 0 THEN

	(* Check battery voltage *)

(* (MB_RegistriLetti[4]) check Livello di Batteria (in millesimi di volt) *)

	IF (MB_RegistriLetti[4]) < LowBattVoltage THEN fBatt := TRUE;
	ELSE fBatt := FALSE;
	END_IF


	Battery(IN:=fBatt);

	IF Battery.EVH  THEN
		LogEv(EL_Wrn,EO_ZTHL,ID,6,' ');
		StatusOK := StatusOK + 1;
	END_IF

	IF Battery.EVL THEN StatusOK := SEL(StatusOK=0, StatusOK-1, 0); END_IF

(* (MB_RegistriLetti[6]) check Temperatura (in decimi di grado centigrado) *)

	(* Check Node temperature *)
	IF (MB_RegistriLetti[6]) < Tmin OR (MB_RegistriLetti[6]) > Tmax THEN
		fTemp := TRUE;
		ERR := TRUE;
	ELSE
		fTemp := FALSE;
		ERR := FALSE;
	END_IF

	Temperature(IN:=fTemp);

	IF Temperature.EVH THEN
		LogEv(EL_Wrn,EO_ZTHL,ID,5,INT_TO_STRING((MB_RegistriLetti[6])));
		Status_Log := 1;
		StatusOK := StatusOK + 1;
	END_IF

	IF Temperature.EVL THEN StatusOK := SEL(StatusOK=0, StatusOK-1, 0); END_IF

END_IF

Alarm(IN:=(StatusOK=0));

IF Alarm.EVH THEN
	Status_Log := 0;
	LogEv(EL_Log,EO_ZTHL,ID,1,'');
END_IF

IF Status_Log = 2 THEN Status_Vis := COLOR_RED;
ELSIF Status_Log = 1 THEN Status_Vis := COLOR_YELLOW;
ELSE Status_Vis := COLOR_GREEN;
END_IF
END_ACTION
ACTION Stm:
CASE state OF
	0:	(* Refresh time manager *)
		ReadTmr(IN:=NOT ReadTmr.Q);
		(*A tempo interrogo il nodo sempre che non ci sia qualcuno che lo sta interrogando in quel momento *)

		IF (ReadTmr.Q AND NodoDaInterrogareMB2=id_locale )OR Refresh_Now AND NOT InibiscoModbusMB2 THEN
			state := 10;
			ReadTmr.PT := T#5s;  (* moreno *)
			Refresh_Now := FALSE;
			InibiscoModbusMB2 := TRUE;
		END_IF

	(**** Leggo le Analogiche a Disposzione  ****)

	10:	(* richiedo lettura Holding Register   *)

		Modbus.MB_Query.SlaveAddress := Address;
		Modbus.MB_Query.FunctionCode := 4;
		ModBus.MB_Query.Read_StartAddress := 0 ;			(* richiedo lettura altri Parametri *)
		ModBus.MB_Query.Read_Quantity := 10;
		ModBus.MB_Start := TRUE;
		state := 20;

	20:	(* Risposta all'interrogazione *)
		IF NOT ModBus.MB_Start   THEN
			VerificaFuctionCode:=ModBus.MB_Resp.FunctionCode;
			VerificaNodoLetto:=ModBus.MB_Resp.SlaveAddress;

			IF ModBus.MB_MASTER.MB_Error<>0 THEN
				state := 300;
			ELSE

				MB_RegistriLetti[0] := ModBus.MB_Resp.Data[0];   	(* Vedi tabella *)
				MB_RegistriLetti[1] := ModBus.MB_Resp.Data[1];		(* Vedi tabella *)
				MB_RegistriLetti[2] := ModBus.MB_Resp.Data[2];		(* Vedi tabella *)
				MB_RegistriLetti[3] := ModBus.MB_Resp.Data[3];		(* Vedi tabella *)
				MB_RegistriLetti[4] := ModBus.MB_Resp.Data[4];		(* Vedi tabella *)
				MB_RegistriLetti[5] := ModBus.MB_Resp.Data[5];		(* Vedi tabella *)
				MB_RegistriLetti[6] := ModBus.MB_Resp.Data[6];		(* Vedi tabella *)
				MB_RegistriLetti[7] := ModBus.MB_Resp.Data[7];		(* Vedi tabella *)
				MB_RegistriLetti[8] := ModBus.MB_Resp.Data[8];		(* Vedi tabella *)
				MB_RegistriLetti[9] := ModBus.MB_Resp.Data[9];		(* Vedi tabella *)
				MB_RegistriLetti[10] := ModBus.MB_Resp.Data[10];		(* Vedi tabella *)
				MB_RegistriLetti[11] := ModBus.MB_Resp.Data[11];		(* Vedi tabella *)
				MB_RegistriLetti[12] := ModBus.MB_Resp.Data[12];		(* Vedi tabella *)
				MB_RegistriLetti[13] := ModBus.MB_Resp.Data[13];		(* Vedi tabella *)

				state := 295;
			END_IF
		END_IF


		295:
		IF NOT ModBus.MB_Start THEN
			IF ModBus.MB_MASTER.MB_Error<>0 THEN (*OR ModBus.MB_MASTER.MB_Error<>0 THEN*)
				state := 300;
			ELSE
				IF fModbusAlr THEN fModbusAlr := FALSE; END_IF
				NodoDaInterrogareMB2:=id_locale+1;
				InibiscoModbusMB2:=FALSE;
				retryErr := 0;
				retry := 0;
				state := 0;
					IF fModbusAlr=FALSE AND ErroreComuModBus=TRUE THEN
						LogEv(EL_Log,EO_CHI,ID,62,'ComunicazioneModBus_OK');
						ErroreComuModBus := FALSE;
				(*	WarningCtr := SEL(WarningCtr=0, WarningCtr-1, 0); *)
					END_IF


			END_IF
		END_IF



	(**** CHECK MODBUS ERROR ****)
	300: 	(* Release MODBUS *)
			InibiscoModbusMB3:=FALSE;
			(* Retries *)
			retry:=retry+1;
			IF retry>3 THEN
				retry:=0;

				(* Verify if slave is dead *)
				IF retryErr < retryErrMaX THEN
					retryErr := retryErr + 1;
				ELSE
					fModbusAlr := TRUE;
					(* Verify ModBus error	*)

					IF fModbusAlr AND ErroreComuModBus=FALSE THEN
						LogEv(EL_Alarm,EO_CHI,ID,61,CONCAT('ErroreModbus_',INT_TO_STRING(ModBus.MB_MASTER.MB_Error)));
						ErroreComuModBus := TRUE;
					END_IF
				END_IF

			END_IF
			Refresh_Now := FALSE;
			InibiscoModbusMB2:=FALSE;
			NodoDaInterrogareMB2:=id_locale+1;
			state:=0;
END_CASE




(* Controllo Time Out Ciclo ModBus *)

TimeOutModBus(In:=state<>0,PT:=t#30s);
IF TimeOutModBus.Q THEN
	State:=0;
	Refresh_Now:=TRUE;  (* Rilancio la lettura del nodo *)
	IF MODBUS.MB_Lock=TRUE THEN MODBUS.MB_Lock:=FALSE;END_IF
	IF InibiscoModbusMB2=TRUE THEN InibiscoModbusMB2:=FALSE;END_IF
END_IF
END_ACTION

(* POU Utils Functions/PLANT_STATUS, ST *)
FUNCTION_BLOCK PLANT_STATUS
VAR_INPUT
	obj_Status		:	WORD;
END_VAR
VAR_OUTPUT
END_VAR
VAR
	PLANT_STATUS	:	WORD;

	Pwm				:	TON := (PT:=T#1s);
END_VAR
CASE plant_Status OF

	0:	(* Plant OK - Everything works well *)
		(*Pwm(IN:=FALSE);	*)						(* Stop timer if running *)
		LAMP_AL := FALSE;						(* Keep the lamp switched off *)

	(*1:	(* Plant in warning *)
		Pwm(IN:= NOT(Pwm.Q));

		IF Pwm.Q THEN
			LAMP_AL := NOT LAMP_AL;				(* Toggle output *)
		END_IF*)

	2:	(* Plant in alarm *)
		(*Pwm(IN:=FALSE);	*)						(* Stop timer if running *)
		LAMP_AL	:= TRUE;						(* Keep the lamp switched on *)

END_CASE

plant_Status := 0;		(* Reset plant status *)
END_FUNCTION_BLOCK
ACTION UpdateStatus:
IF plant_Status = 2 THEN

	RETURN;					(* If plant already in alarm condition do nothing *)

ELSE

		IF obj_Status <> 0 THEN
			plant_Status := obj_Status;			(* If plant in warning/normal condition and current object in alarm, update plant status *)
		END_IF
END_IF
END_ACTION

(* POU PLC_WDT, ST *)
FUNCTION PLC_WDT: DWORD VAR_INPUT dwEvent: DWORD; dwFilter: DWORD; dwOwner: DWORD; END_VAR
LogEv(EL_AlarmStop,EO_SYS,1,10,'Watchdog');
END_FUNCTION

(* POU Utils Functions/RAW16TOHEXSTR, ST *)
FUNCTION RAW16TOHEXSTR : STRING(128)
VAR_INPUT
	pData: POINTER TO BYTE;
	DataLen: BYTE;
END_VAR
VAR
	pt: POINTER TO BYTE;
	xl: BYTE;
END_VAR
pt:=ADR(RAW16TOHEXSTR);
xl:=0;

WHILE DataLen>0 AND xl<120 DO

	pData:=pData+1;

	pt^ := (pData^ / 16#10) + 48 + (((pData^ / 16#10)/10)*7);
	pt:=pt+1;
	pt^ := (pData^ AND 16#0F)  + 48 + (((pData^ AND 16#0F)/10)*7);
	pt:=pt+1;

	pData:=pData-1;

	pt^ := (pData^ / 16#10) + 48 + (((pData^ / 16#10)/10)*7);
	pt:=pt+1;
	pt^ := (pData^ AND 16#0F)  + 48 + (((pData^ AND 16#0F)/10)*7);
	pt:=pt+1;

	xl:=xl+4;

	DataLen:=DataLen-2;
	pData:=pData+2;

END_WHILE

pt^:=0;
END_FUNCTION

(* POU Utils Functions/RAWTOHEXSTR, ST *)
FUNCTION RAWTOHEXSTR : STRING(128)
VAR_INPUT
	pData: POINTER TO BYTE;
	DataLen: BYTE;
END_VAR
VAR
	pt: POINTER TO BYTE;
	xl: BYTE;
END_VAR
pt:=ADR(RAWTOHEXSTR);

xl:=2;

WHILE DataLen>0 AND xl<128 DO

	pt^ := (pData^ / 16#10) + 48 + (((pData^ / 16#10)/10)*7);
	pt:=pt+1;
	pt^ := (pData^ AND 16#0F)  + 48 + (((pData^ AND 16#0F)/10)*7);
	pt:=pt+1;

	xl:=xl+2;

	DataLen:=DataLen-1;
	pData:=pData+1;

END_WHILE

pt^:=0;
END_FUNCTION

(* POU Utils/RTC_Update, ST *)
FUNCTION RTC_Update : BOOL
VAR
	T: DT;
	TS: STRING;
	TS2: STRING;
	Hour: BYTE;
	Minute: BYTE;
END_VAR
(* Get RTC time *)
T:=SysRtcGetTime(TRUE);
Sys.Time_CT_DT:=T;
(* Calculate variables *)
TS:=DT_TO_STRING(T);
Sys.Time_LogString:=DELETE(STR:=TS, LEN:=3, POS:=1);
TS2:=MID(STR:=TS, LEN:=4, POS:= 4); Sys.Time_Year 	:=STRING_TO_WORD(TS2);
TS2:=MID(STR:=TS, LEN:=2, POS:= 9); Sys.Time_Month	:=STRING_TO_BYTE(TS2);
TS2:=MID(STR:=TS, LEN:=2, POS:=12); Sys.Time_Day  	:=STRING_TO_BYTE(TS2);
Sys.Time_CT_Day:=(32*(Sys.Time_Month-1)+Sys.Time_Day-1);
TS2:=MID(STR:=TS, LEN:=2, POS:=15); Hour			:=STRING_TO_BYTE(TS2);
TS2:=MID(STR:=TS, LEN:=2, POS:=18); Minute		 	:=STRING_TO_BYTE(TS2);
Sys.Time_Hour := Hour;
Sys.Time_Minute := Minute;
Sys.Time_CT_Quarter:=Hour*4+(Minute/15);
END_FUNCTION

(* POU Utils Functions/SHIFT_ARRAY, ST *)
FUNCTION SHIFT_ARRAY : BOOL
VAR_INPUT
	pData	:	POINTER TO ARRAY [1..2] OF WORD;
	Size	:	BYTE;
END_VAR
VAR
	pNew	:	POINTER TO WORD;
	i		:	BYTE;
END_VAR
(* Shift right *)
FOR i:=1 TO (Size-1) BY 1 DO

	(*pNew := pData + 1;*)
	pData^[i] := pData^[i+1];
	(*pData := pData + 1;*)

END_FOR
END_FUNCTION

(* Visualisation PLC_VISU
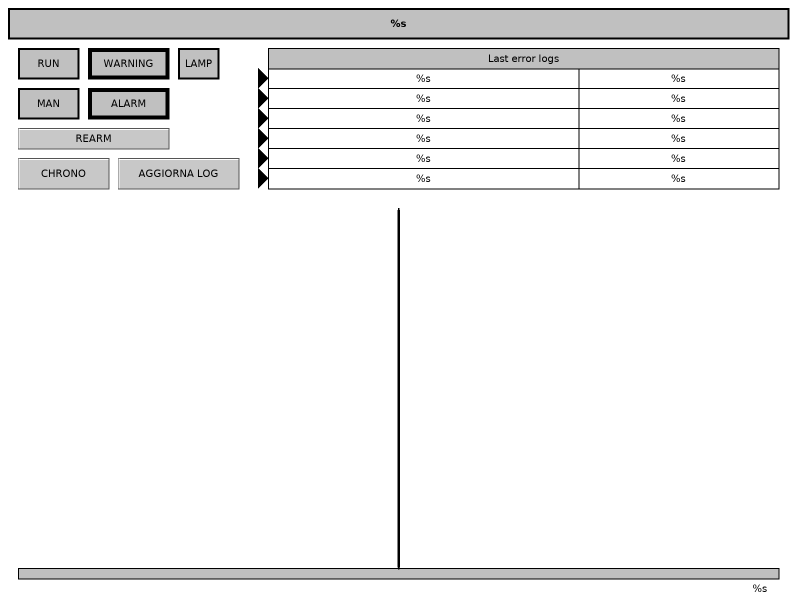
rectangle at (10,10)-(791,41): text "%s"; shows .Plant_NAME
rectangle at (530,580)-(771,601): text "%s"; shows Sys.Time_LogString
rounded rectangle at (20,50)-(81,81): text "RUN"; alarm colour if NOT Mode_Manual; runs INTERN ASSIGN Mode_Manual:=(FALSE)
rounded rectangle at (20,90)-(81,121): text "MAN"; alarm colour if Mode_Manual; runs INTERN ASSIGN Mode_Manual:=(TRUE)
rectangle at (580,70)-(781,91): text "%s"; shows Sys.LastLogs_Msg[0]
polygon at (260,170)-(270,190): invisible if Sys.LastLogs_Idx<>0
rectangle at (580,90)-(781,111): text "%s"; shows Sys.LastLogs_Msg[1]
polygon at (260,70)-(270,90): invisible if Sys.LastLogs_Idx<>1
rectangle at (580,110)-(781,131): text "%s"; shows Sys.LastLogs_Msg[2]
polygon at (260,90)-(270,110): invisible if Sys.LastLogs_Idx<>2
rectangle at (580,130)-(781,151): text "%s"; shows Sys.LastLogs_Msg[3]
polygon at (260,110)-(270,130): invisible if Sys.LastLogs_Idx<>3
rectangle at (580,150)-(781,171): text "%s"; shows Sys.LastLogs_Msg[4]
polygon at (260,130)-(270,150): invisible if Sys.LastLogs_Idx<>4
rectangle at (580,170)-(781,191): text "%s"; shows Sys.LastLogs_Msg[5]
polygon at (260,150)-(270,170): invisible if Sys.LastLogs_Idx<>5
rectangle at (270,70)-(581,91): text "%s"; shows Sys.LastLogs_Dat[0]
rectangle at (270,90)-(581,111): text "%s"; shows Sys.LastLogs_Dat[1]
rectangle at (270,110)-(581,131): text "%s"; shows Sys.LastLogs_Dat[2]
rectangle at (270,130)-(581,151): text "%s"; shows Sys.LastLogs_Dat[3]
rectangle at (270,150)-(581,171): text "%s"; shows Sys.LastLogs_Dat[4]
rectangle at (270,170)-(581,191): text "%s"; shows Sys.LastLogs_Dat[5]
rectangle at (90,90)-(171,121): text "ALARM"; alarm colour if Sys.Alarm; runs INTERN ASSIGN Mode_Manual:=(FALSE)
rectangle at (90,50)-(171,81): text "WARNING"; alarm colour if Sys.Warning; runs INTERN ASSIGN Mode_Manual:=(TRUE)
button at (20,130)-(171,151): text "REARM"; runs INTERN ASSIGN Sys.Alarm:=(FALSE);INTERN ASSIGN Sys.Warning:=(FALSE)
rectangle at (270,50)-(781,71): text "Last error logs"
rounded rectangle at (180,50)-(221,81): text "LAMP"; alarm colour if LAMP_AL
button at (20,160)-(111,191): text "CHRONO"; opens VIS_CHONOEDITOR
button at (120,160)-(241,191): text "AGGIORNA LOG"; taps .AggiornaLog
2 more shapes without text or variables
*)

(* Visualisation VIS_CHONOEDITOR
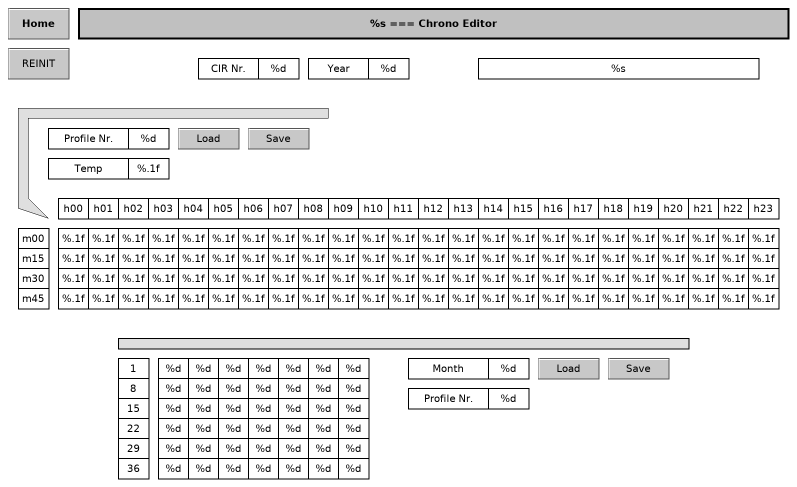
rectangle at (200,60)-(261,81): text "CIR Nr."
rectangle at (260,60)-(301,81): text "%d"; shows CronEd.CN_Sel; alarm colour if CronEd.CN_Sel<>CronEd.CN_Act; editable 1..250
rectangle at (50,130)-(131,151): text "Profile Nr."
rectangle at (130,130)-(171,151): text "%d"; shows CronEd.PR_Sel; alarm colour if CronEd.PR_Sel<>CronEd.PR_Act; editable 1..10
rectangle at (50,160)-(131,181): text "Temp"
rectangle at (130,160)-(171,181): text "%.1f"; shows CronEd.PR_TT; editable
button at (180,130)-(241,151): text "Load"; toggles CronEd.PR_Load
button at (250,130)-(311,151): text "Save"; toggles CronEd.PR_Save
rectangle at (20,230)-(51,251): text "m00"
rectangle at (20,250)-(51,271): text "m15"
rectangle at (20,270)-(51,291): text "m30"
rectangle at (20,290)-(51,311): text "m45"
rectangle at (80,10)-(791,41): text "%s === Chrono Editor"; shows .Plant_NAME
button at (10,10)-(71,41): text "Home"; opens PLC_VISU
rounded rectangle at (60,230)-(91,251): text "%.1f"; shows WORD_TO_REAL(CronEd.PR.Setpoint[0])/10; runs INTERN ASSIGN CronEd.PR.Setpoint[0]:=(REAL_TO_WORD(CronEd.PR_TT*10))
rounded rectangle at (60,250)-(91,271): text "%.1f"; shows WORD_TO_REAL(CronEd.PR.Setpoint[1])/10; runs INTERN ASSIGN CronEd.PR.Setpoint[1]:=(REAL_TO_WORD(CronEd.PR_TT*10))
rounded rectangle at (60,270)-(91,291): text "%.1f"; shows WORD_TO_REAL(CronEd.PR.Setpoint[2])/10; runs INTERN ASSIGN CronEd.PR.Setpoint[2]:=(REAL_TO_WORD(CronEd.PR_TT*10))
rounded rectangle at (60,290)-(91,311): text "%.1f"; shows WORD_TO_REAL(CronEd.PR.Setpoint[3])/10; runs INTERN ASSIGN CronEd.PR.Setpoint[3]:=(REAL_TO_WORD(CronEd.PR_TT*10))
rectangle at (60,200)-(91,221): text "h00"; runs INTERN ASSIGN CronEd.PR.Setpoint[0]:=(REAL_TO_WORD(CronEd.PR_TT*10));INTERN ASSIGN CronEd.PR.Setpoint[1]:=(REAL_TO_WORD(CronEd.PR_TT*10));INTERN ASSIGN CronEd.PR.Setpoint[2]:=(REAL_TO_WORD(CronEd.PR_TT*10));INTERN ASSIGN CronEd.PR.Setpoint[3]:=(REAL_TO_WORD(CronEd.PR_TT*10))
rounded rectangle at (90,230)-(121,251): text "%.1f"; shows WORD_TO_REAL(CronEd.PR.Setpoint[4])/10; runs INTERN ASSIGN CronEd.PR.Setpoint[4]:=(REAL_TO_WORD(CronEd.PR_TT*10))
rounded rectangle at (90,250)-(121,271): text "%.1f"; shows WORD_TO_REAL(CronEd.PR.Setpoint[5])/10; runs INTERN ASSIGN CronEd.PR.Setpoint[5]:=(REAL_TO_WORD(CronEd.PR_TT*10))
rounded rectangle at (90,270)-(121,291): text "%.1f"; shows WORD_TO_REAL(CronEd.PR.Setpoint[6])/10; runs INTERN ASSIGN CronEd.PR.Setpoint[6]:=(REAL_TO_WORD(CronEd.PR_TT*10))
rounded rectangle at (90,290)-(121,311): text "%.1f"; shows WORD_TO_REAL(CronEd.PR.Setpoint[7])/10; runs INTERN ASSIGN CronEd.PR.Setpoint[7]:=(REAL_TO_WORD(CronEd.PR_TT*10))
rectangle at (90,200)-(121,221): text "h01"; runs INTERN ASSIGN CronEd.PR.Setpoint[4]:=(REAL_TO_WORD(CronEd.PR_TT*10));INTERN ASSIGN CronEd.PR.Setpoint[5]:=(REAL_TO_WORD(CronEd.PR_TT*10));INTERN ASSIGN CronEd.PR.Setpoint[6]:=(REAL_TO_WORD(CronEd.PR_TT*10));INTERN ASSIGN CronEd.PR.Setpoint[7]:=(REAL_TO_WORD(CronEd.PR_TT*10))
rounded rectangle at (120,230)-(151,251): text "%.1f"; shows WORD_TO_REAL(CronEd.PR.Setpoint[8])/10; runs INTERN ASSIGN CronEd.PR.Setpoint[8]:=(REAL_TO_WORD(CronEd.PR_TT*10))
rounded rectangle at (120,250)-(151,271): text "%.1f"; shows WORD_TO_REAL(CronEd.PR.Setpoint[9])/10; runs INTERN ASSIGN CronEd.PR.Setpoint[9]:=(REAL_TO_WORD(CronEd.PR_TT*10))
rounded rectangle at (120,270)-(151,291): text "%.1f"; shows WORD_TO_REAL(CronEd.PR.Setpoint[10])/10; runs INTERN ASSIGN CronEd.PR.Setpoint[10]:=(REAL_TO_WORD(CronEd.PR_TT*10))
rounded rectangle at (120,290)-(151,311): text "%.1f"; shows WORD_TO_REAL(CronEd.PR.Setpoint[11])/10; runs INTERN ASSIGN CronEd.PR.Setpoint[11]:=(REAL_TO_WORD(CronEd.PR_TT*10))
rectangle at (120,200)-(151,221): text "h02"; runs INTERN ASSIGN CronEd.PR.Setpoint[8]:=(REAL_TO_WORD(CronEd.PR_TT*10));INTERN ASSIGN CronEd.PR.Setpoint[9]:=(REAL_TO_WORD(CronEd.PR_TT*10));INTERN ASSIGN CronEd.PR.Setpoint[10]:=(REAL_TO_WORD(CronEd.PR_TT*10));INTERN ASSIGN CronEd.PR.Setpoint[11]:=(REAL_TO_WORD(CronEd.PR_TT*10))
rounded rectangle at (150,230)-(181,251): text "%.1f"; shows WORD_TO_REAL(CronEd.PR.Setpoint[12])/10; runs INTERN ASSIGN CronEd.PR.Setpoint[12]:=(REAL_TO_WORD(CronEd.PR_TT*10))
rounded rectangle at (150,250)-(181,271): text "%.1f"; shows WORD_TO_REAL(CronEd.PR.Setpoint[13])/10; runs INTERN ASSIGN CronEd.PR.Setpoint[13]:=(REAL_TO_WORD(CronEd.PR_TT*10))
rounded rectangle at (150,270)-(181,291): text "%.1f"; shows WORD_TO_REAL(CronEd.PR.Setpoint[14])/10; runs INTERN ASSIGN CronEd.PR.Setpoint[14]:=(REAL_TO_WORD(CronEd.PR_TT*10))
rounded rectangle at (150,290)-(181,311): text "%.1f"; shows WORD_TO_REAL(CronEd.PR.Setpoint[15])/10; runs INTERN ASSIGN CronEd.PR.Setpoint[15]:=(REAL_TO_WORD(CronEd.PR_TT*10))
rectangle at (150,200)-(181,221): text "h03"; runs INTERN ASSIGN CronEd.PR.Setpoint[15]:=(REAL_TO_WORD(CronEd.PR_TT*10));INTERN ASSIGN CronEd.PR.Setpoint[14]:=(REAL_TO_WORD(CronEd.PR_TT*10));INTERN ASSIGN CronEd.PR.Setpoint[13]:=(REAL_TO_WORD(CronEd.PR_TT*10));INTERN ASSIGN CronEd.PR.Setpoint[12]:=(REAL_TO_WORD(CronEd.PR_TT*10))
rounded rectangle at (180,230)-(211,251): text "%.1f"; shows WORD_TO_REAL(CronEd.PR.Setpoint[16])/10; runs INTERN ASSIGN CronEd.PR.Setpoint[16]:=(REAL_TO_WORD(CronEd.PR_TT*10))
rounded rectangle at (180,250)-(211,271): text "%.1f"; shows WORD_TO_REAL(CronEd.PR.Setpoint[17])/10; runs INTERN ASSIGN CronEd.PR.Setpoint[17]:=(REAL_TO_WORD(CronEd.PR_TT*10))
rounded rectangle at (180,270)-(211,291): text "%.1f"; shows WORD_TO_REAL(CronEd.PR.Setpoint[18])/10; runs INTERN ASSIGN CronEd.PR.Setpoint[18]:=(REAL_TO_WORD(CronEd.PR_TT*10))
rounded rectangle at (180,290)-(211,311): text "%.1f"; shows WORD_TO_REAL(CronEd.PR.Setpoint[19])/10; runs INTERN ASSIGN CronEd.PR.Setpoint[19]:=(REAL_TO_WORD(CronEd.PR_TT*10))
rectangle at (180,200)-(211,221): text "h04"; runs INTERN ASSIGN CronEd.PR.Setpoint[19]:=(REAL_TO_WORD(CronEd.PR_TT*10));INTERN ASSIGN CronEd.PR.Setpoint[18]:=(REAL_TO_WORD(CronEd.PR_TT*10));INTERN ASSIGN CronEd.PR.Setpoint[17]:=(REAL_TO_WORD(CronEd.PR_TT*10));INTERN ASSIGN CronEd.PR.Setpoint[16]:=(REAL_TO_WORD(CronEd.PR_TT*10))
rounded rectangle at (210,230)-(241,251): text "%.1f"; shows WORD_TO_REAL(CronEd.PR.Setpoint[20])/10; runs INTERN ASSIGN CronEd.PR.Setpoint[20]:=(REAL_TO_WORD(CronEd.PR_TT*10))
rounded rectangle at (210,250)-(241,271): text "%.1f"; shows WORD_TO_REAL(CronEd.PR.Setpoint[21])/10; runs INTERN ASSIGN CronEd.PR.Setpoint[21]:=(REAL_TO_WORD(CronEd.PR_TT*10))
rounded rectangle at (210,270)-(241,291): text "%.1f"; shows WORD_TO_REAL(CronEd.PR.Setpoint[22])/10; runs INTERN ASSIGN CronEd.PR.Setpoint[22]:=(REAL_TO_WORD(CronEd.PR_TT*10))
rounded rectangle at (210,290)-(241,311): text "%.1f"; shows WORD_TO_REAL(CronEd.PR.Setpoint[23])/10; runs INTERN ASSIGN CronEd.PR.Setpoint[23]:=(REAL_TO_WORD(CronEd.PR_TT*10))
rectangle at (210,200)-(241,221): text "h05"; runs INTERN ASSIGN CronEd.PR.Setpoint[23]:=(REAL_TO_WORD(CronEd.PR_TT*10));INTERN ASSIGN CronEd.PR.Setpoint[22]:=(REAL_TO_WORD(CronEd.PR_TT*10));INTERN ASSIGN CronEd.PR.Setpoint[21]:=(REAL_TO_WORD(CronEd.PR_TT*10));INTERN ASSIGN CronEd.PR.Setpoint[20]:=(REAL_TO_WORD(CronEd.PR_TT*10))
rounded rectangle at (240,230)-(271,251): text "%.1f"; shows WORD_TO_REAL(CronEd.PR.Setpoint[24])/10; runs INTERN ASSIGN CronEd.PR.Setpoint[24]:=(REAL_TO_WORD(CronEd.PR_TT*10))
rounded rectangle at (240,250)-(271,271): text "%.1f"; shows WORD_TO_REAL(CronEd.PR.Setpoint[25])/10; runs INTERN ASSIGN CronEd.PR.Setpoint[25]:=(REAL_TO_WORD(CronEd.PR_TT*10))
rounded rectangle at (240,270)-(271,291): text "%.1f"; shows WORD_TO_REAL(CronEd.PR.Setpoint[26])/10; runs INTERN ASSIGN CronEd.PR.Setpoint[26]:=(REAL_TO_WORD(CronEd.PR_TT*10))
rounded rectangle at (240,290)-(271,311): text "%.1f"; shows WORD_TO_REAL(CronEd.PR.Setpoint[27])/10; runs INTERN ASSIGN CronEd.PR.Setpoint[27]:=(REAL_TO_WORD(CronEd.PR_TT*10))
rectangle at (240,200)-(271,221): text "h06"; runs INTERN ASSIGN CronEd.PR.Setpoint[27]:=(REAL_TO_WORD(CronEd.PR_TT*10));INTERN ASSIGN CronEd.PR.Setpoint[26]:=(REAL_TO_WORD(CronEd.PR_TT*10));INTERN ASSIGN CronEd.PR.Setpoint[25]:=(REAL_TO_WORD(CronEd.PR_TT*10));INTERN ASSIGN CronEd.PR.Setpoint[24]:=(REAL_TO_WORD(CronEd.PR_TT*10))
rounded rectangle at (270,230)-(301,251): text "%.1f"; shows WORD_TO_REAL(CronEd.PR.Setpoint[28])/10; runs INTERN ASSIGN CronEd.PR.Setpoint[28]:=(REAL_TO_WORD(CronEd.PR_TT*10))
rounded rectangle at (270,250)-(301,271): text "%.1f"; shows WORD_TO_REAL(CronEd.PR.Setpoint[29])/10; runs INTERN ASSIGN CronEd.PR.Setpoint[29]:=(REAL_TO_WORD(CronEd.PR_TT*10))
rounded rectangle at (270,270)-(301,291): text "%.1f"; shows WORD_TO_REAL(CronEd.PR.Setpoint[30])/10; runs INTERN ASSIGN CronEd.PR.Setpoint[30]:=(REAL_TO_WORD(CronEd.PR_TT*10))
rounded rectangle at (270,290)-(301,311): text "%.1f"; shows WORD_TO_REAL(CronEd.PR.Setpoint[31])/10; runs INTERN ASSIGN CronEd.PR.Setpoint[31]:=(REAL_TO_WORD(CronEd.PR_TT*10))
rectangle at (270,200)-(301,221): text "h07"; runs INTERN ASSIGN CronEd.PR.Setpoint[31]:=(REAL_TO_WORD(CronEd.PR_TT*10));INTERN ASSIGN CronEd.PR.Setpoint[30]:=(REAL_TO_WORD(CronEd.PR_TT*10));INTERN ASSIGN CronEd.PR.Setpoint[29]:=(REAL_TO_WORD(CronEd.PR_TT*10));INTERN ASSIGN CronEd.PR.Setpoint[28]:=(REAL_TO_WORD(CronEd.PR_TT*10))
rounded rectangle at (300,230)-(331,251): text "%.1f"; shows WORD_TO_REAL(CronEd.PR.Setpoint[32])/10; runs INTERN ASSIGN CronEd.PR.Setpoint[32]:=(REAL_TO_WORD(CronEd.PR_TT*10))
rounded rectangle at (300,250)-(331,271): text "%.1f"; shows WORD_TO_REAL(CronEd.PR.Setpoint[33])/10; runs INTERN ASSIGN CronEd.PR.Setpoint[33]:=(REAL_TO_WORD(CronEd.PR_TT*10))
rounded rectangle at (300,270)-(331,291): text "%.1f"; shows WORD_TO_REAL(CronEd.PR.Setpoint[34])/10; runs INTERN ASSIGN CronEd.PR.Setpoint[34]:=(REAL_TO_WORD(CronEd.PR_TT*10))
rounded rectangle at (300,290)-(331,311): text "%.1f"; shows WORD_TO_REAL(CronEd.PR.Setpoint[35])/10; runs INTERN ASSIGN CronEd.PR.Setpoint[35]:=(REAL_TO_WORD(CronEd.PR_TT*10))
rectangle at (300,200)-(331,221): text "h08"; runs INTERN ASSIGN CronEd.PR.Setpoint[35]:=(REAL_TO_WORD(CronEd.PR_TT*10));INTERN ASSIGN CronEd.PR.Setpoint[34]:=(REAL_TO_WORD(CronEd.PR_TT*10));INTERN ASSIGN CronEd.PR.Setpoint[33]:=(REAL_TO_WORD(CronEd.PR_TT*10));INTERN ASSIGN CronEd.PR.Setpoint[32]:=(REAL_TO_WORD(CronEd.PR_TT*10))
rounded rectangle at (330,230)-(361,251): text "%.1f"; shows WORD_TO_REAL(CronEd.PR.Setpoint[36])/10; runs INTERN ASSIGN CronEd.PR.Setpoint[36]:=(REAL_TO_WORD(CronEd.PR_TT*10))
rounded rectangle at (330,250)-(361,271): text "%.1f"; shows WORD_TO_REAL(CronEd.PR.Setpoint[37])/10; runs INTERN ASSIGN CronEd.PR.Setpoint[37]:=(REAL_TO_WORD(CronEd.PR_TT*10))
rounded rectangle at (330,270)-(361,291): text "%.1f"; shows WORD_TO_REAL(CronEd.PR.Setpoint[38])/10; runs INTERN ASSIGN CronEd.PR.Setpoint[38]:=(REAL_TO_WORD(CronEd.PR_TT*10))
rounded rectangle at (330,290)-(361,311): text "%.1f"; shows WORD_TO_REAL(CronEd.PR.Setpoint[39])/10; runs INTERN ASSIGN CronEd.PR.Setpoint[39]:=(REAL_TO_WORD(CronEd.PR_TT*10))
rectangle at (330,200)-(361,221): text "h09"; runs INTERN ASSIGN CronEd.PR.Setpoint[39]:=(REAL_TO_WORD(CronEd.PR_TT*10));INTERN ASSIGN CronEd.PR.Setpoint[38]:=(REAL_TO_WORD(CronEd.PR_TT*10));INTERN ASSIGN CronEd.PR.Setpoint[37]:=(REAL_TO_WORD(CronEd.PR_TT*10));INTERN ASSIGN CronEd.PR.Setpoint[36]:=(REAL_TO_WORD(CronEd.PR_TT*10))
rounded rectangle at (360,230)-(391,251): text "%.1f"; shows WORD_TO_REAL(CronEd.PR.Setpoint[40])/10; runs INTERN ASSIGN CronEd.PR.Setpoint[40]:=(REAL_TO_WORD(CronEd.PR_TT*10))
rounded rectangle at (360,250)-(391,271): text "%.1f"; shows WORD_TO_REAL(CronEd.PR.Setpoint[41])/10; runs INTERN ASSIGN CronEd.PR.Setpoint[41]:=(REAL_TO_WORD(CronEd.PR_TT*10))
rounded rectangle at (360,270)-(391,291): text "%.1f"; shows WORD_TO_REAL(CronEd.PR.Setpoint[42])/10; runs INTERN ASSIGN CronEd.PR.Setpoint[42]:=(REAL_TO_WORD(CronEd.PR_TT*10))
rounded rectangle at (360,290)-(391,311): text "%.1f"; shows WORD_TO_REAL(CronEd.PR.Setpoint[43])/10; runs INTERN ASSIGN CronEd.PR.Setpoint[43]:=(REAL_TO_WORD(CronEd.PR_TT*10))
rectangle at (360,200)-(391,221): text "h10"; runs INTERN ASSIGN CronEd.PR.Setpoint[43]:=(REAL_TO_WORD(CronEd.PR_TT*10));INTERN ASSIGN CronEd.PR.Setpoint[42]:=(REAL_TO_WORD(CronEd.PR_TT*10));INTERN ASSIGN CronEd.PR.Setpoint[41]:=(REAL_TO_WORD(CronEd.PR_TT*10));INTERN ASSIGN CronEd.PR.Setpoint[40]:=(REAL_TO_WORD(CronEd.PR_TT*10))
rounded rectangle at (390,230)-(421,251): text "%.1f"; shows WORD_TO_REAL(CronEd.PR.Setpoint[44])/10; runs INTERN ASSIGN CronEd.PR.Setpoint[44]:=(REAL_TO_WORD(CronEd.PR_TT*10))
rounded rectangle at (390,250)-(421,271): text "%.1f"; shows WORD_TO_REAL(CronEd.PR.Setpoint[45])/10; runs INTERN ASSIGN CronEd.PR.Setpoint[45]:=(REAL_TO_WORD(CronEd.PR_TT*10))
rounded rectangle at (390,270)-(421,291): text "%.1f"; shows WORD_TO_REAL(CronEd.PR.Setpoint[46])/10; runs INTERN ASSIGN CronEd.PR.Setpoint[46]:=(REAL_TO_WORD(CronEd.PR_TT*10))
rounded rectangle at (390,290)-(421,311): text "%.1f"; shows WORD_TO_REAL(CronEd.PR.Setpoint[47])/10; runs INTERN ASSIGN CronEd.PR.Setpoint[47]:=(REAL_TO_WORD(CronEd.PR_TT*10))
rectangle at (390,200)-(421,221): text "h11"; runs INTERN ASSIGN CronEd.PR.Setpoint[47]:=(REAL_TO_WORD(CronEd.PR_TT*10));INTERN ASSIGN CronEd.PR.Setpoint[46]:=(REAL_TO_WORD(CronEd.PR_TT*10));INTERN ASSIGN CronEd.PR.Setpoint[45]:=(REAL_TO_WORD(CronEd.PR_TT*10));INTERN ASSIGN CronEd.PR.Setpoint[44]:=(REAL_TO_WORD(CronEd.PR_TT*10))
rounded rectangle at (420,230)-(451,251): text "%.1f"; shows WORD_TO_REAL(CronEd.PR.Setpoint[48])/10; runs INTERN ASSIGN CronEd.PR.Setpoint[48]:=(REAL_TO_WORD(CronEd.PR_TT*10))
rounded rectangle at (420,250)-(451,271): text "%.1f"; shows WORD_TO_REAL(CronEd.PR.Setpoint[49])/10; runs INTERN ASSIGN CronEd.PR.Setpoint[49]:=(REAL_TO_WORD(CronEd.PR_TT*10))
rounded rectangle at (420,270)-(451,291): text "%.1f"; shows WORD_TO_REAL(CronEd.PR.Setpoint[50])/10; runs INTERN ASSIGN CronEd.PR.Setpoint[50]:=(REAL_TO_WORD(CronEd.PR_TT*10))
rounded rectangle at (420,290)-(451,311): text "%.1f"; shows WORD_TO_REAL(CronEd.PR.Setpoint[51])/10; runs INTERN ASSIGN CronEd.PR.Setpoint[51]:=(REAL_TO_WORD(CronEd.PR_TT*10))
rectangle at (420,200)-(451,221): text "h12"; runs INTERN ASSIGN CronEd.PR.Setpoint[51]:=(REAL_TO_WORD(CronEd.PR_TT*10));INTERN ASSIGN CronEd.PR.Setpoint[50]:=(REAL_TO_WORD(CronEd.PR_TT*10));INTERN ASSIGN CronEd.PR.Setpoint[49]:=(REAL_TO_WORD(CronEd.PR_TT*10));INTERN ASSIGN CronEd.PR.Setpoint[48]:=(REAL_TO_WORD(CronEd.PR_TT*10))
rounded rectangle at (450,230)-(481,251): text "%.1f"; shows WORD_TO_REAL(CronEd.PR.Setpoint[52])/10; runs INTERN ASSIGN CronEd.PR.Setpoint[52]:=(REAL_TO_WORD(CronEd.PR_TT*10))
rounded rectangle at (450,250)-(481,271): text "%.1f"; shows WORD_TO_REAL(CronEd.PR.Setpoint[53])/10; runs INTERN ASSIGN CronEd.PR.Setpoint[53]:=(REAL_TO_WORD(CronEd.PR_TT*10))
rounded rectangle at (450,270)-(481,291): text "%.1f"; shows WORD_TO_REAL(CronEd.PR.Setpoint[54])/10; runs INTERN ASSIGN CronEd.PR.Setpoint[54]:=(REAL_TO_WORD(CronEd.PR_TT*10))
rounded rectangle at (450,290)-(481,311): text "%.1f"; shows WORD_TO_REAL(CronEd.PR.Setpoint[55])/10; runs INTERN ASSIGN CronEd.PR.Setpoint[55]:=(REAL_TO_WORD(CronEd.PR_TT*10))
rectangle at (450,200)-(481,221): text "h13"; runs INTERN ASSIGN CronEd.PR.Setpoint[55]:=(REAL_TO_WORD(CronEd.PR_TT*10));INTERN ASSIGN CronEd.PR.Setpoint[54]:=(REAL_TO_WORD(CronEd.PR_TT*10));INTERN ASSIGN CronEd.PR.Setpoint[53]:=(REAL_TO_WORD(CronEd.PR_TT*10));INTERN ASSIGN CronEd.PR.Setpoint[52]:=(REAL_TO_WORD(CronEd.PR_TT*10))
rounded rectangle at (480,230)-(511,251): text "%.1f"; shows WORD_TO_REAL(CronEd.PR.Setpoint[56])/10; runs INTERN ASSIGN CronEd.PR.Setpoint[56]:=(REAL_TO_WORD(CronEd.PR_TT*10))
rounded rectangle at (480,250)-(511,271): text "%.1f"; shows WORD_TO_REAL(CronEd.PR.Setpoint[57])/10; runs INTERN ASSIGN CronEd.PR.Setpoint[57]:=(REAL_TO_WORD(CronEd.PR_TT*10))
rounded rectangle at (480,270)-(511,291): text "%.1f"; shows WORD_TO_REAL(CronEd.PR.Setpoint[58])/10; runs INTERN ASSIGN CronEd.PR.Setpoint[58]:=(REAL_TO_WORD(CronEd.PR_TT*10))
rounded rectangle at (480,290)-(511,311): text "%.1f"; shows WORD_TO_REAL(CronEd.PR.Setpoint[59])/10; runs INTERN ASSIGN CronEd.PR.Setpoint[59]:=(REAL_TO_WORD(CronEd.PR_TT*10))
rectangle at (480,200)-(511,221): text "h14"; runs INTERN ASSIGN CronEd.PR.Setpoint[59]:=(REAL_TO_WORD(CronEd.PR_TT*10));INTERN ASSIGN CronEd.PR.Setpoint[58]:=(REAL_TO_WORD(CronEd.PR_TT*10));INTERN ASSIGN CronEd.PR.Setpoint[57]:=(REAL_TO_WORD(CronEd.PR_TT*10));INTERN ASSIGN CronEd.PR.Setpoint[56]:=(REAL_TO_WORD(CronEd.PR_TT*10))
rounded rectangle at (510,230)-(541,251): text "%.1f"; shows WORD_TO_REAL(CronEd.PR.Setpoint[60])/10; runs INTERN ASSIGN CronEd.PR.Setpoint[60]:=(REAL_TO_WORD(CronEd.PR_TT*10))
rounded rectangle at (510,250)-(541,271): text "%.1f"; shows WORD_TO_REAL(CronEd.PR.Setpoint[61])/10; runs INTERN ASSIGN CronEd.PR.Setpoint[61]:=(REAL_TO_WORD(CronEd.PR_TT*10))
rounded rectangle at (510,270)-(541,291): text "%.1f"; shows WORD_TO_REAL(CronEd.PR.Setpoint[62])/10; runs INTERN ASSIGN CronEd.PR.Setpoint[62]:=(REAL_TO_WORD(CronEd.PR_TT*10))
rounded rectangle at (510,290)-(541,311): text "%.1f"; shows WORD_TO_REAL(CronEd.PR.Setpoint[63])/10; runs INTERN ASSIGN CronEd.PR.Setpoint[63]:=(REAL_TO_WORD(CronEd.PR_TT*10))
rectangle at (510,200)-(541,221): text "h15"; runs INTERN ASSIGN CronEd.PR.Setpoint[63]:=(REAL_TO_WORD(CronEd.PR_TT*10));INTERN ASSIGN CronEd.PR.Setpoint[62]:=(REAL_TO_WORD(CronEd.PR_TT*10));INTERN ASSIGN CronEd.PR.Setpoint[61]:=(REAL_TO_WORD(CronEd.PR_TT*10));INTERN ASSIGN CronEd.PR.Setpoint[60]:=(REAL_TO_WORD(CronEd.PR_TT*10))
rounded rectangle at (540,230)-(571,251): text "%.1f"; shows WORD_TO_REAL(CronEd.PR.Setpoint[64])/10; runs INTERN ASSIGN CronEd.PR.Setpoint[64]:=(REAL_TO_WORD(CronEd.PR_TT*10))
rounded rectangle at (540,250)-(571,271): text "%.1f"; shows WORD_TO_REAL(CronEd.PR.Setpoint[65])/10; runs INTERN ASSIGN CronEd.PR.Setpoint[65]:=(REAL_TO_WORD(CronEd.PR_TT*10))
rounded rectangle at (540,270)-(571,291): text "%.1f"; shows WORD_TO_REAL(CronEd.PR.Setpoint[66])/10; runs INTERN ASSIGN CronEd.PR.Setpoint[66]:=(REAL_TO_WORD(CronEd.PR_TT*10))
rounded rectangle at (540,290)-(571,311): text "%.1f"; shows WORD_TO_REAL(CronEd.PR.Setpoint[67])/10; runs INTERN ASSIGN CronEd.PR.Setpoint[67]:=(REAL_TO_WORD(CronEd.PR_TT*10))
rectangle at (540,200)-(571,221): text "h16"; runs INTERN ASSIGN CronEd.PR.Setpoint[67]:=(REAL_TO_WORD(CronEd.PR_TT*10));INTERN ASSIGN CronEd.PR.Setpoint[66]:=(REAL_TO_WORD(CronEd.PR_TT*10));INTERN ASSIGN CronEd.PR.Setpoint[65]:=(REAL_TO_WORD(CronEd.PR_TT*10));INTERN ASSIGN CronEd.PR.Setpoint[64]:=(REAL_TO_WORD(CronEd.PR_TT*10))
rounded rectangle at (570,230)-(601,251): text "%.1f"; shows WORD_TO_REAL(CronEd.PR.Setpoint[68])/10; runs INTERN ASSIGN CronEd.PR.Setpoint[68]:=(REAL_TO_WORD(CronEd.PR_TT*10))
rounded rectangle at (570,250)-(601,271): text "%.1f"; shows WORD_TO_REAL(CronEd.PR.Setpoint[69])/10; runs INTERN ASSIGN CronEd.PR.Setpoint[69]:=(REAL_TO_WORD(CronEd.PR_TT*10))
rounded rectangle at (570,270)-(601,291): text "%.1f"; shows WORD_TO_REAL(CronEd.PR.Setpoint[70])/10; runs INTERN ASSIGN CronEd.PR.Setpoint[70]:=(REAL_TO_WORD(CronEd.PR_TT*10))
rounded rectangle at (570,290)-(601,311): text "%.1f"; shows WORD_TO_REAL(CronEd.PR.Setpoint[71])/10; runs INTERN ASSIGN CronEd.PR.Setpoint[71]:=(REAL_TO_WORD(CronEd.PR_TT*10))
rectangle at (570,200)-(601,221): text "h17"; runs INTERN ASSIGN CronEd.PR.Setpoint[71]:=(REAL_TO_WORD(CronEd.PR_TT*10));INTERN ASSIGN CronEd.PR.Setpoint[70]:=(REAL_TO_WORD(CronEd.PR_TT*10));INTERN ASSIGN CronEd.PR.Setpoint[69]:=(REAL_TO_WORD(CronEd.PR_TT*10));INTERN ASSIGN CronEd.PR.Setpoint[68]:=(REAL_TO_WORD(CronEd.PR_TT*10))
rounded rectangle at (600,230)-(631,251): text "%.1f"; shows WORD_TO_REAL(CronEd.PR.Setpoint[72])/10; runs INTERN ASSIGN CronEd.PR.Setpoint[72]:=(REAL_TO_WORD(CronEd.PR_TT*10))
rounded rectangle at (600,250)-(631,271): text "%.1f"; shows WORD_TO_REAL(CronEd.PR.Setpoint[73])/10; runs INTERN ASSIGN CronEd.PR.Setpoint[73]:=(REAL_TO_WORD(CronEd.PR_TT*10))
rounded rectangle at (600,270)-(631,291): text "%.1f"; shows WORD_TO_REAL(CronEd.PR.Setpoint[74])/10; runs INTERN ASSIGN CronEd.PR.Setpoint[74]:=(REAL_TO_WORD(CronEd.PR_TT*10))
rounded rectangle at (600,290)-(631,311): text "%.1f"; shows WORD_TO_REAL(CronEd.PR.Setpoint[75])/10; runs INTERN ASSIGN CronEd.PR.Setpoint[75]:=(REAL_TO_WORD(CronEd.PR_TT*10))
rectangle at (600,200)-(631,221): text "h18"; runs INTERN ASSIGN CronEd.PR.Setpoint[75]:=(REAL_TO_WORD(CronEd.PR_TT*10));INTERN ASSIGN CronEd.PR.Setpoint[74]:=(REAL_TO_WORD(CronEd.PR_TT*10));INTERN ASSIGN CronEd.PR.Setpoint[73]:=(REAL_TO_WORD(CronEd.PR_TT*10));INTERN ASSIGN CronEd.PR.Setpoint[72]:=(REAL_TO_WORD(CronEd.PR_TT*10))
rounded rectangle at (630,230)-(661,251): text "%.1f"; shows WORD_TO_REAL(CronEd.PR.Setpoint[76])/10; runs INTERN ASSIGN CronEd.PR.Setpoint[76]:=(REAL_TO_WORD(CronEd.PR_TT*10))
rounded rectangle at (630,250)-(661,271): text "%.1f"; shows WORD_TO_REAL(CronEd.PR.Setpoint[77])/10; runs INTERN ASSIGN CronEd.PR.Setpoint[77]:=(REAL_TO_WORD(CronEd.PR_TT*10))
rounded rectangle at (630,270)-(661,291): text "%.1f"; shows WORD_TO_REAL(CronEd.PR.Setpoint[78])/10; runs INTERN ASSIGN CronEd.PR.Setpoint[78]:=(REAL_TO_WORD(CronEd.PR_TT*10))
rounded rectangle at (630,290)-(661,311): text "%.1f"; shows WORD_TO_REAL(CronEd.PR.Setpoint[79])/10; runs INTERN ASSIGN CronEd.PR.Setpoint[79]:=(REAL_TO_WORD(CronEd.PR_TT*10))
rectangle at (630,200)-(661,221): text "h19"; runs INTERN ASSIGN CronEd.PR.Setpoint[79]:=(REAL_TO_WORD(CronEd.PR_TT*10));INTERN ASSIGN CronEd.PR.Setpoint[78]:=(REAL_TO_WORD(CronEd.PR_TT*10));INTERN ASSIGN CronEd.PR.Setpoint[77]:=(REAL_TO_WORD(CronEd.PR_TT*10));INTERN ASSIGN CronEd.PR.Setpoint[76]:=(REAL_TO_WORD(CronEd.PR_TT*10))
rounded rectangle at (660,230)-(691,251): text "%.1f"; shows WORD_TO_REAL(CronEd.PR.Setpoint[80])/10; runs INTERN ASSIGN CronEd.PR.Setpoint[80]:=(REAL_TO_WORD(CronEd.PR_TT*10))
rounded rectangle at (660,250)-(691,271): text "%.1f"; shows WORD_TO_REAL(CronEd.PR.Setpoint[81])/10; runs INTERN ASSIGN CronEd.PR.Setpoint[81]:=(REAL_TO_WORD(CronEd.PR_TT*10))
rounded rectangle at (660,270)-(691,291): text "%.1f"; shows WORD_TO_REAL(CronEd.PR.Setpoint[82])/10; runs INTERN ASSIGN CronEd.PR.Setpoint[82]:=(REAL_TO_WORD(CronEd.PR_TT*10))
rounded rectangle at (660,290)-(691,311): text "%.1f"; shows WORD_TO_REAL(CronEd.PR.Setpoint[83])/10; runs INTERN ASSIGN CronEd.PR.Setpoint[83]:=(REAL_TO_WORD(CronEd.PR_TT*10))
rectangle at (660,200)-(691,221): text "h20"; runs INTERN ASSIGN CronEd.PR.Setpoint[83]:=(REAL_TO_WORD(CronEd.PR_TT*10));INTERN ASSIGN CronEd.PR.Setpoint[82]:=(REAL_TO_WORD(CronEd.PR_TT*10));INTERN ASSIGN CronEd.PR.Setpoint[81]:=(REAL_TO_WORD(CronEd.PR_TT*10));INTERN ASSIGN CronEd.PR.Setpoint[80]:=(REAL_TO_WORD(CronEd.PR_TT*10))
rounded rectangle at (690,230)-(721,251): text "%.1f"; shows WORD_TO_REAL(CronEd.PR.Setpoint[84])/10; runs INTERN ASSIGN CronEd.PR.Setpoint[84]:=(REAL_TO_WORD(CronEd.PR_TT*10))
rounded rectangle at (690,250)-(721,271): text "%.1f"; shows WORD_TO_REAL(CronEd.PR.Setpoint[85])/10; runs INTERN ASSIGN CronEd.PR.Setpoint[85]:=(REAL_TO_WORD(CronEd.PR_TT*10))
rounded rectangle at (690,270)-(721,291): text "%.1f"; shows WORD_TO_REAL(CronEd.PR.Setpoint[86])/10; runs INTERN ASSIGN CronEd.PR.Setpoint[86]:=(REAL_TO_WORD(CronEd.PR_TT*10))
rounded rectangle at (690,290)-(721,311): text "%.1f"; shows WORD_TO_REAL(CronEd.PR.Setpoint[87])/10; runs INTERN ASSIGN CronEd.PR.Setpoint[87]:=(REAL_TO_WORD(CronEd.PR_TT*10))
rectangle at (690,200)-(721,221): text "h21"; runs INTERN ASSIGN CronEd.PR.Setpoint[87]:=(REAL_TO_WORD(CronEd.PR_TT*10));INTERN ASSIGN CronEd.PR.Setpoint[86]:=(REAL_TO_WORD(CronEd.PR_TT*10));INTERN ASSIGN CronEd.PR.Setpoint[85]:=(REAL_TO_WORD(CronEd.PR_TT*10));INTERN ASSIGN CronEd.PR.Setpoint[84]:=(REAL_TO_WORD(CronEd.PR_TT*10))
rounded rectangle at (720,230)-(751,251): text "%.1f"; shows WORD_TO_REAL(CronEd.PR.Setpoint[88])/10; runs INTERN ASSIGN CronEd.PR.Setpoint[88]:=(REAL_TO_WORD(CronEd.PR_TT*10))
rounded rectangle at (720,250)-(751,271): text "%.1f"; shows WORD_TO_REAL(CronEd.PR.Setpoint[89])/10; runs INTERN ASSIGN CronEd.PR.Setpoint[89]:=(REAL_TO_WORD(CronEd.PR_TT*10))
rounded rectangle at (720,270)-(751,291): text "%.1f"; shows WORD_TO_REAL(CronEd.PR.Setpoint[90])/10; runs INTERN ASSIGN CronEd.PR.Setpoint[90]:=(REAL_TO_WORD(CronEd.PR_TT*10))
rounded rectangle at (720,290)-(751,311): text "%.1f"; shows WORD_TO_REAL(CronEd.PR.Setpoint[91])/10; runs INTERN ASSIGN CronEd.PR.Setpoint[91]:=(REAL_TO_WORD(CronEd.PR_TT*10))
rectangle at (720,200)-(751,221): text "h22"; runs INTERN ASSIGN CronEd.PR.Setpoint[91]:=(REAL_TO_WORD(CronEd.PR_TT*10));INTERN ASSIGN CronEd.PR.Setpoint[90]:=(REAL_TO_WORD(CronEd.PR_TT*10));INTERN ASSIGN CronEd.PR.Setpoint[89]:=(REAL_TO_WORD(CronEd.PR_TT*10));INTERN ASSIGN CronEd.PR.Setpoint[88]:=(REAL_TO_WORD(CronEd.PR_TT*10))
rounded rectangle at (750,230)-(781,251): text "%.1f"; shows WORD_TO_REAL(CronEd.PR.Setpoint[92])/10; runs INTERN ASSIGN CronEd.PR.Setpoint[92]:=(REAL_TO_WORD(CronEd.PR_TT*10))
rounded rectangle at (750,250)-(781,271): text "%.1f"; shows WORD_TO_REAL(CronEd.PR.Setpoint[93])/10; runs INTERN ASSIGN CronEd.PR.Setpoint[93]:=(REAL_TO_WORD(CronEd.PR_TT*10))
rounded rectangle at (750,270)-(781,291): text "%.1f"; shows WORD_TO_REAL(CronEd.PR.Setpoint[94])/10; runs INTERN ASSIGN CronEd.PR.Setpoint[94]:=(REAL_TO_WORD(CronEd.PR_TT*10))
rounded rectangle at (750,290)-(781,311): text "%.1f"; shows WORD_TO_REAL(CronEd.PR.Setpoint[95])/10; runs INTERN ASSIGN CronEd.PR.Setpoint[95]:=(REAL_TO_WORD(CronEd.PR_TT*10))
rectangle at (750,200)-(781,221): text "h23"; runs INTERN ASSIGN CronEd.PR.Setpoint[95]:=(REAL_TO_WORD(CronEd.PR_TT*10));INTERN ASSIGN CronEd.PR.Setpoint[94]:=(REAL_TO_WORD(CronEd.PR_TT*10));INTERN ASSIGN CronEd.PR.Setpoint[93]:=(REAL_TO_WORD(CronEd.PR_TT*10));INTERN ASSIGN CronEd.PR.Setpoint[92]:=(REAL_TO_WORD(CronEd.PR_TT*10))
rectangle at (410,360)-(491,381): text "Month"
rectangle at (490,360)-(531,381): text "%d"; shows CronEd.CA_Sel; alarm colour if CronEd.CA_Sel<>CronEd.CA_Act; editable 1..12
rectangle at (410,390)-(491,411): text "Profile Nr."
rectangle at (490,390)-(531,411): text "%d"; shows CronEd.CA_TPR; editable 0..10
button at (540,360)-(601,381): text "Load"; toggles CronEd.CA_Load
button at (610,360)-(671,381): text "Save"; toggles CronEd.CA_Save
rounded rectangle at (160,360)-(191,381): text "%d"; shows CronEd.CA.Profile[0]; invisible if CronEd.CA_DayF>0; alarm colour if CronEd.CA.Profile[0]=0; runs INTERN ASSIGN CronEd.CA.Profile[0]:=(CronEd.CA_TPR)
rectangle at (120,360)-(151,381): text "1"
rounded rectangle at (190,360)-(221,381): text "%d"; shows CronEd.CA.Profile[1]; invisible if CronEd.CA_DayF>1; alarm colour if CronEd.CA.Profile[1]=0; runs INTERN ASSIGN CronEd.CA.Profile[1]:=(CronEd.CA_TPR)
rounded rectangle at (220,360)-(251,381): text "%d"; shows CronEd.CA.Profile[2]; invisible if CronEd.CA_DayF>2; alarm colour if CronEd.CA.Profile[2]=0; runs INTERN ASSIGN CronEd.CA.Profile[2]:=(CronEd.CA_TPR)
rounded rectangle at (250,360)-(281,381): text "%d"; shows CronEd.CA.Profile[3]; invisible if CronEd.CA_DayF>3; alarm colour if CronEd.CA.Profile[3]=0; runs INTERN ASSIGN CronEd.CA.Profile[3]:=(CronEd.CA_TPR)
rounded rectangle at (280,360)-(311,381): text "%d"; shows CronEd.CA.Profile[4]; invisible if CronEd.CA_DayF>4; alarm colour if CronEd.CA.Profile[4]=0; runs INTERN ASSIGN CronEd.CA.Profile[4]:=(CronEd.CA_TPR)
rounded rectangle at (310,360)-(341,381): text "%d"; shows CronEd.CA.Profile[5]; invisible if CronEd.CA_DayF>5; alarm colour if CronEd.CA.Profile[5]=0; runs INTERN ASSIGN CronEd.CA.Profile[5]:=(CronEd.CA_TPR)
rounded rectangle at (340,360)-(371,381): text "%d"; shows CronEd.CA.Profile[6]; alarm colour if CronEd.CA.Profile[6]=0; runs INTERN ASSIGN CronEd.CA.Profile[6]:=(CronEd.CA_TPR)
rounded rectangle at (160,380)-(191,401): text "%d"; shows CronEd.CA.Profile[7]; alarm colour if CronEd.CA.Profile[7]=0; runs INTERN ASSIGN CronEd.CA.Profile[7]:=(CronEd.CA_TPR)
rectangle at (120,380)-(151,401): text "8"
rounded rectangle at (190,380)-(221,401): text "%d"; shows CronEd.CA.Profile[8]; alarm colour if CronEd.CA.Profile[8]=0; runs INTERN ASSIGN CronEd.CA.Profile[8]:=(CronEd.CA_TPR)
rounded rectangle at (220,380)-(251,401): text "%d"; shows CronEd.CA.Profile[9]; alarm colour if CronEd.CA.Profile[9]=0; runs INTERN ASSIGN CronEd.CA.Profile[9]:=(CronEd.CA_TPR)
rounded rectangle at (250,380)-(281,401): text "%d"; shows CronEd.CA.Profile[10]; alarm colour if CronEd.CA.Profile[10]=0; runs INTERN ASSIGN CronEd.CA.Profile[10]:=(CronEd.CA_TPR)
rounded rectangle at (280,380)-(311,401): text "%d"; shows CronEd.CA.Profile[11]; alarm colour if CronEd.CA.Profile[11]=0; runs INTERN ASSIGN CronEd.CA.Profile[11]:=(CronEd.CA_TPR)
rounded rectangle at (310,380)-(341,401): text "%d"; shows CronEd.CA.Profile[12]; alarm colour if CronEd.CA.Profile[12]=0; runs INTERN ASSIGN CronEd.CA.Profile[12]:=(CronEd.CA_TPR)
rounded rectangle at (340,380)-(371,401): text "%d"; shows CronEd.CA.Profile[13]; alarm colour if CronEd.CA.Profile[13]=0; runs INTERN ASSIGN CronEd.CA.Profile[13]:=(CronEd.CA_TPR)
rounded rectangle at (160,400)-(191,421): text "%d"; shows CronEd.CA.Profile[14]; alarm colour if CronEd.CA.Profile[14]=0; runs INTERN ASSIGN CronEd.CA.Profile[14]:=(CronEd.CA_TPR)
rectangle at (120,400)-(151,421): text "15"
rounded rectangle at (190,400)-(221,421): text "%d"; shows CronEd.CA.Profile[15]; alarm colour if CronEd.CA.Profile[15]=0; runs INTERN ASSIGN CronEd.CA.Profile[15]:=(CronEd.CA_TPR)
rounded rectangle at (220,400)-(251,421): text "%d"; shows CronEd.CA.Profile[16]; alarm colour if CronEd.CA.Profile[16]=0; runs INTERN ASSIGN CronEd.CA.Profile[16]:=(CronEd.CA_TPR)
rounded rectangle at (250,400)-(281,421): text "%d"; shows CronEd.CA.Profile[17]; alarm colour if CronEd.CA.Profile[17]=0; runs INTERN ASSIGN CronEd.CA.Profile[17]:=(CronEd.CA_TPR)
rounded rectangle at (280,400)-(311,421): text "%d"; shows CronEd.CA.Profile[18]; alarm colour if CronEd.CA.Profile[18]=0; runs INTERN ASSIGN CronEd.CA.Profile[18]:=(CronEd.CA_TPR)
rounded rectangle at (310,400)-(341,421): text "%d"; shows CronEd.CA.Profile[19]; alarm colour if CronEd.CA.Profile[19]=0; runs INTERN ASSIGN CronEd.CA.Profile[19]:=(CronEd.CA_TPR)
rounded rectangle at (340,400)-(371,421): text "%d"; shows CronEd.CA.Profile[20]; alarm colour if CronEd.CA.Profile[20]=0; runs INTERN ASSIGN CronEd.CA.Profile[20]:=(CronEd.CA_TPR)
rounded rectangle at (160,420)-(191,441): text "%d"; shows CronEd.CA.Profile[21]; alarm colour if CronEd.CA.Profile[21]=0; runs INTERN ASSIGN CronEd.CA.Profile[21]:=(CronEd.CA_TPR)
rectangle at (120,420)-(151,441): text "22"
rounded rectangle at (190,420)-(221,441): text "%d"; shows CronEd.CA.Profile[22]; alarm colour if CronEd.CA.Profile[22]=0; runs INTERN ASSIGN CronEd.CA.Profile[22]:=(CronEd.CA_TPR)
rounded rectangle at (220,420)-(251,441): text "%d"; shows CronEd.CA.Profile[23]; alarm colour if CronEd.CA.Profile[23]=0; runs INTERN ASSIGN CronEd.CA.Profile[23]:=(CronEd.CA_TPR)
rounded rectangle at (250,420)-(281,441): text "%d"; shows CronEd.CA.Profile[24]; alarm colour if CronEd.CA.Profile[24]=0; runs INTERN ASSIGN CronEd.CA.Profile[24]:=(CronEd.CA_TPR)
rounded rectangle at (280,420)-(311,441): text "%d"; shows CronEd.CA.Profile[25]; alarm colour if CronEd.CA.Profile[25]=0; runs INTERN ASSIGN CronEd.CA.Profile[25]:=(CronEd.CA_TPR)
rounded rectangle at (310,420)-(341,441): text "%d"; shows CronEd.CA.Profile[26]; alarm colour if CronEd.CA.Profile[26]=0; runs INTERN ASSIGN CronEd.CA.Profile[26]:=(CronEd.CA_TPR)
rounded rectangle at (340,420)-(371,441): text "%d"; shows CronEd.CA.Profile[27]; alarm colour if CronEd.CA.Profile[27]=0; runs INTERN ASSIGN CronEd.CA.Profile[27]:=(CronEd.CA_TPR)
rounded rectangle at (160,440)-(191,461): text "%d"; shows CronEd.CA.Profile[28]; alarm colour if CronEd.CA.Profile[28]=0; runs INTERN ASSIGN CronEd.CA.Profile[28]:=(CronEd.CA_TPR)
rectangle at (120,440)-(151,461): text "29"
rounded rectangle at (190,440)-(221,461): text "%d"; shows CronEd.CA.Profile[29]; alarm colour if CronEd.CA.Profile[29]=0; runs INTERN ASSIGN CronEd.CA.Profile[29]:=(CronEd.CA_TPR)
rounded rectangle at (220,440)-(251,461): text "%d"; shows CronEd.CA.Profile[30]; alarm colour if CronEd.CA.Profile[30]=0; runs INTERN ASSIGN CronEd.CA.Profile[30]:=(CronEd.CA_TPR)
rounded rectangle at (250,440)-(281,461): text "%d"; shows CronEd.CA.Profile[31]; alarm colour if CronEd.CA.Profile[31]=0; runs INTERN ASSIGN CronEd.CA.Profile[31]:=(CronEd.CA_TPR)
rounded rectangle at (280,440)-(311,461): text "%d"; shows CronEd.CA.Profile[32]; invisible if CronEd.CA_DayL<32; alarm colour if CronEd.CA.Profile[32]=0; runs INTERN ASSIGN CronEd.CA.Profile[32]:=(CronEd.CA_TPR)
rounded rectangle at (310,440)-(341,461): text "%d"; shows CronEd.CA.Profile[33]; invisible if CronEd.CA_DayL<33; alarm colour if CronEd.CA.Profile[33]=0; runs INTERN ASSIGN CronEd.CA.Profile[33]:=(CronEd.CA_TPR)
rounded rectangle at (340,440)-(371,461): text "%d"; shows CronEd.CA.Profile[34]; invisible if CronEd.CA_DayL<34; alarm colour if CronEd.CA.Profile[34]=0; runs INTERN ASSIGN CronEd.CA.Profile[34]:=(CronEd.CA_TPR)
rounded rectangle at (160,460)-(191,481): text "%d"; shows CronEd.CA.Profile[35]; invisible if CronEd.CA_DayL<35; alarm colour if CronEd.CA.Profile[35]=0; runs INTERN ASSIGN CronEd.CA.Profile[35]:=(CronEd.CA_TPR)
rectangle at (120,460)-(151,481): text "36"; invisible if CronEd.CA_DayL<35
rounded rectangle at (190,460)-(221,481): text "%d"; shows CronEd.CA.Profile[36]; invisible if CronEd.CA_DayL<36; alarm colour if CronEd.CA.Profile[36]=0; runs INTERN ASSIGN CronEd.CA.Profile[36]:=(CronEd.CA_TPR)
rounded rectangle at (220,460)-(251,481): text "%d"; shows CronEd.CA.Profile[37]; invisible if CronEd.CA_DayL<37; alarm colour if CronEd.CA.Profile[37]=0; runs INTERN ASSIGN CronEd.CA.Profile[37]:=(CronEd.CA_TPR)
rounded rectangle at (250,460)-(281,481): text "%d"; shows CronEd.CA.Profile[38]; invisible if CronEd.CA_DayL<38; alarm colour if CronEd.CA.Profile[38]=0; runs INTERN ASSIGN CronEd.CA.Profile[38]:=(CronEd.CA_TPR)
rounded rectangle at (280,460)-(311,481): text "%d"; shows CronEd.CA.Profile[39]; invisible if CronEd.CA_DayL<39; alarm colour if CronEd.CA.Profile[39]=0; runs INTERN ASSIGN CronEd.CA.Profile[39]:=(CronEd.CA_TPR)
rounded rectangle at (310,460)-(341,481): text "%d"; shows CronEd.CA.Profile[40]; invisible if CronEd.CA_DayL<40; alarm colour if CronEd.CA.Profile[40]=0; runs INTERN ASSIGN CronEd.CA.Profile[40]:=(CronEd.CA_TPR)
rounded rectangle at (340,460)-(371,481): text "%d"; shows CronEd.CA.Profile[41]; invisible if CronEd.CA_DayL<41; alarm colour if CronEd.CA.Profile[41]=0; runs INTERN ASSIGN CronEd.CA.Profile[41]:=(CronEd.CA_TPR)
rectangle at (310,60)-(371,81): text "Year"
rectangle at (370,60)-(411,81): text "%d"; shows CronEd.CN_YSel; alarm colour if CronEd.CN_YSel<>CronEd.CN_YAct; editable 2000..2100
rectangle at (480,60)-(761,81): text "%s"; shows CronEd.Message
button at (10,50)-(71,81): text "REINIT"; runs INTERN ASSIGN THER01.InitOK:=(FALSE);INTERN ASSIGN THER02.InitOK:=(FALSE);INTERN ASSIGN THER03.InitOK:=(FALSE);INTERN ASSIGN THER04.InitOK:=(FALSE);INTERN ASSIGN THER05.InitOK:=(FALSE);INTERN ASSIGN THER06.InitOK:=(FALSE)
2 more shapes without text or variables
*)
